C05474=1017.752,-121.815,388.715,-23.943,21.711,-44.591
C05475=1017.748,-122.143,388.737,-23.942,21.712,-44.597
C05476=1017.744,-122.471,388.759,-23.942,21.713,-44.601
C05477=1017.741,-122.799,388.781,-23.941,21.713,-44.606
C05478=1017.737,-123.128,388.803,-23.940,21.714,-44.610
C05479=1017.733,-123.456,388.826,-23.940,21.714,-44.615
C05480=1017.729,-123.785,388.848,-23.939,21.715,-44.620
C05481=1017.725,-124.112,388.871,-23.939,21.715,-44.625
C05482=1017.721,-124.441,388.893,-23.938,21.716,-44.628
C05483=1017.717,-124.769,388.915,-23.937,21.717,-44.634
C05484=1017.713,-125.097,388.937,-23.937,21.717,-44.638
C05485=1017.709,-125.425,388.959,-23.936,21.717,-44.643
C05486=1017.706,-125.754,388.981,-23.936,21.719,-44.647
C05487=1017.702,-126.082,389.003,-23.935,21.719,-44.652
C05488=1017.697,-126.409,389.026,-23.935,21.720,-44.657
C05489=1017.693,-126.737,389.048,-23.934,21.720,-44.662
C05490=1017.689,-127.066,389.070,-23.933,21.720,-44.667
C05491=1017.686,-127.394,389.092,-23.933,21.721,-44.671
C05492=1017.682,-127.722,389.114,-23.932,21.721,-44.676
C05493=1017.677,-128.050,389.136,-23.931,21.722,-44.680
C05494=1017.674,-128.378,389.158,-23.931,21.723,-44.686
C05495=1017.670,-128.706,389.180,-23.930,21.723,-44.689
C05496=1017.665,-129.034,389.202,-23.929,21.723,-44.695
C05497=1017.661,-129.362,389.224,-23.929,21.725,-44.699
C05498=1017.657,-129.690,389.246,-23.928,21.724,-44.704
C05499=1017.653,-130.018,389.268,-23.928,21.726,-44.708
C05500=1017.649,-130.346,389.290,-23.927,21.726,-44.713
C05501=1017.644,-130.674,389.312,-23.927,21.726,-44.717
C05502=1017.641,-131.002,389.334,-23.926,21.727,-44.723
C05503=1017.636,-131.331,389.356,-23.926,21.728,-44.726
C05504=1017.632,-131.659,389.378,-23.925,21.728,-44.732
C05505=1017.627,-131.986,389.400,-23.924,21.729,-44.736
C05506=1017.622,-132.314,389.422,-23.924,21.729,-44.741
C05507=1017.619,-132.643,389.444,-23.923,21.730,-44.745
C05508=1017.614,-132.971,389.465,-23.922,21.731,-44.750
C05509=1017.610,-133.299,389.488,-23.922,21.731,-44.754
C05510=1017.606,-133.626,389.510,-23.921,21.731,-44.759
C05511=1017.601,-133.954,389.531,-23.921,21.732,-44.763
C05512=1017.986,-133.926,389.292,-23.921,21.732,-44.763
C05513=1017.990,-133.599,389.270,-23.921,21.731,-44.759
C05514=1017.994,-133.271,389.248,-23.922,21.731,-44.754
C05515=1017.999,-132.943,389.226,-23.922,21.731,-44.750
C05516=1018.002,-132.614,389.204,-23.923,21.730,-44.745
C05517=1018.007,-132.287,389.182,-23.924,21.729,-44.741
C05518=1018.011,-131.959,389.161,-23.924,21.729,-44.736
C05519=1018.015,-131.630,389.139,-23.925,21.728,-44.732
C05520=1018.020,-131.303,389.117,-23.926,21.728,-44.726
C05521=1018.024,-130.975,389.094,-23.926,21.727,-44.723
C05522=1018.028,-130.647,389.073,-23.927,21.726,-44.717
C05523=1018.032,-130.319,389.051,-23.927,21.726,-44.713
C05524=1018.036,-129.990,389.029,-23.928,21.726,-44.708
C05525=1018.040,-129.662,389.007,-23.928,21.724,-44.704
C05526=1018.044,-129.334,388.985,-23.929,21.725,-44.699
C05527=1018.049,-129.006,388.964,-23.929,21.723,-44.695
C05528=1018.053,-128.679,388.941,-23.930,21.723,-44.689
C05529=1018.057,-128.350,388.919,-23.931,21.723,-44.686
C05530=1018.060,-128.022,388.897,-23.931,21.722,-44.680
C05531=1018.065,-127.694,388.875,-23.932,21.721,-44.676
C05532=1018.068,-127.367,388.853,-23.933,21.721,-44.671
C05533=1018.072,-127.038,388.831,-23.933,21.720,-44.667
C05534=1018.076,-126.710,388.809,-23.934,21.720,-44.662
C05535=1018.080,-126.382,388.788,-23.935,21.720,-44.657
C05536=1018.084,-126.054,388.766,-23.935,21.719,-44.652
C05537=1018.088,-125.726,388.743,-23.936,21.719,-44.647
C05538=1018.092,-125.398,388.721,-23.936,21.717,-44.643
C05539=1018.095,-125.070,388.699,-23.937,21.717,-44.638
C05540=1018.099,-124.741,388.676,-23.937,21.717,-44.634
C05541=1018.103,-124.413,388.654,-23.938,21.716,-44.628
C05542=1018.107,-124.085,388.632,-23.939,21.715,-44.625
C05543=1018.111,-123.757,388.610,-23.939,21.715,-44.620
C05544=1018.114,-123.428,388.588,-23.940,21.714,-44.615
C05545=1018.118,-123.100,388.566,-23.940,21.714,-44.610
C05546=1018.122,-122.772,388.544,-23.941,21.713,-44.606
C05547=1018.126,-122.444,388.522,-23.942,21.713,-44.601
C05548=1018.129,-122.115,388.500,-23.942,21.712,-44.597
C05549=1018.132,-121.787,388.477,-23.943,21.711,-44.591
C05550=1018.136,-121.459,388.455,-23.944,21.711,-44.586
C05551=1018.140,-121.130,388.433,-23.944,21.710,-44.582
C05552=1018.144,-120.802,388.411,-23.945,21.710,-44.577
C05553=1018.148,-120.474,388.389,-23.945,21.709,-44.573
C05554=1018.151,-120.145,388.366,-23.946,21.709,-44.568
C05555=1018.154,-119.817,388.344,-23.946,21.708,-44.564
C05556=1018.158,-119.489,388.322,-23.947,21.707,-44.558
C05557=1018.161,-119.160,388.299,-23.948,21.707,-44.554
C05558=1018.165,-118.832,388.277,-23.948,21.707,-44.549
C05559=1018.169,-118.504,388.255,-23.949,21.705,-44.545
C05560=1018.172,-118.175,388.232,-23.949,21.705,-44.540
C05561=1018.175,-117.847,388.210,-23.950,21.705,-44.535
C05562=1018.179,-117.518,388.187,-23.951,21.704,-44.531
C05563=1018.182,-117.190,388.165,-23.951,21.704,-44.525
C05564=1018.185,-116.862,388.142,-23.952,21.703,-44.521
C05565=1018.189,-116.533,388.120,-23.953,21.703,-44.516
C05566=1018.192,-116.205,388.098,-23.953,21.701,-44.512
C05567=1018.196,-115.876,388.076,-23.954,21.701,-44.507
C05568=1018.199,-115.548,388.053,-23.954,21.701,-44.503
C05569=1018.202,-115.219,388.030,-23.955,21.700,-44.497
C05570=1018.206,-114.891,388.008,-23.956,21.700,-44.492
C05571=1018.209,-114.562,387.985,-23.956,21.699,-44.488
C05572=1018.212,-114.234,387.963,-23.957,21.699,-44.483
C05573=1018.215,-113.905,387.940,-23.957,21.698,-44.479
C05574=1018.218,-113.576,387.919,-23.958,21.697,-44.473
C05575=1018.221,-113.248,387.896,-23.958,21.697,-44.470
C05576=1018.224,-112.919,387.873,-23.959,21.696,-44.464
C05577=1018.228,-112.590,387.850,-23.960,21.696,-44.459
C05578=1018.231,-112.261,387.827,-23.960,21.695,-44.455
C05579=1018.234,-111.933,387.805,-23.961,21.695,-44.449
C05580=1018.237,-111.604,387.782,-23.962,21.694,-44.446
C05581=1018.241,-111.276,387.760,-23.962,21.693,-44.440
C05582=1018.244,-110.947,387.738,-23.963,21.693,-44.436
C05583=1018.247,-110.618,387.715,-23.963,21.692,-44.431
C05584=1018.250,-110.289,387.692,-23.964,21.692,-44.426
C05585=1018.253,-109.960,387.669,-23.965,21.691,-44.422
C05586=1018.256,-109.632,387.646,-23.965,21.691,-44.416
C05587=1018.258,-109.302,387.624,-23.966,21.690,-44.412
C05588=1018.261,-108.974,387.602,-23.967,21.689,-44.407
C05589=1018.265,-108.645,387.578,-23.967,21.689,-44.402
C05590=1018.268,-108.316,387.556,-23.968,21.689,-44.398
C05591=1018.270,-107.987,387.532,-23.969,21.688,-44.392
C05592=1018.273,-107.658,387.511,-23.969,21.687,-44.388
C05593=1018.276,-107.329,387.488,-23.970,21.687,-44.383
C05594=1018.280,-107.000,387.465,-23.971,21.687,-44.378
C05595=1018.282,-106.671,387.441,-23.971,21.685,-44.374
C05596=1018.285,-106.342,387.419,-23.972,21.685,-44.368
C05597=1018.288,-106.013,387.397,-23.972,21.685,-44.365
C05598=1018.291,-105.684,387.373,-23.973,21.684,-44.359
C05599=1018.294,-105.355,387.350,-23.974,21.684,-44.354
C05600=1018.296,-105.027,387.328,-23.974,21.683,-44.350
C05601=1018.299,-104.699,387.305,-23.975,21.683,-44.344
C05602=1018.302,-104.370,387.282,-23.975,21.681,-44.340
C05603=1018.304,-104.043,387.259,-23.976,21.681,-44.335
C05604=1018.308,-103.716,387.237,-23.976,21.681,-44.331
C05605=1018.310,-103.389,387.214,-23.977,21.680,-44.326
C05606=1018.313,-103.062,387.191,-23.978,21.680,-44.320
C05607=1018.316,-102.736,387.169,-23.978,21.679,-44.316
C05608=1018.317,-102.411,387.146,-23.979,21.679,-44.311
C05609=1018.321,-102.085,387.123,-23.980,21.678,-44.307
C05610=1018.323,-101.762,387.100,-23.980,21.677,-44.302
C05611=1018.325,-101.437,387.078,-23.981,21.677,-44.298
C05612=1018.328,-101.113,387.055,-23.981,21.676,-44.292
C05613=1018.331,-100.790,387.033,-23.982,21.676,-44.287
C05614=1018.333,-100.468,387.010,-23.983,21.675,-44.283
C05615=1018.336,-100.146,386.987,-23.983,21.675,-44.278
C05616=1018.338,-99.824,386.965,-23.984,21.674,-44.274
C05617=1018.341,-99.502,386.942,-23.985,21.673,-44.268
C05618=1018.343,-99.181,386.920,-23.985,21.673,-44.265
C05619=1018.345,-98.860,386.898,-23.986,21.673,-44.260
C05620=1018.348,-98.539,386.874,-23.986,21.671,-44.255
C05621=1018.351,-98.217,386.852,-23.987,21.672,-44.250
C05622=1018.353,-97.897,386.829,-23.987,21.670,-44.246
C05623=1018.355,-97.576,386.807,-23.988,21.670,-44.241
C05624=1018.358,-97.255,386.784,-23.989,21.670,-44.236
C05625=1018.360,-96.934,386.762,-23.989,21.669,-44.231
C05626=1018.361,-96.613,386.739,-23.990,21.669,-44.226
C05627=1018.364,-96.291,386.716,-23.991,21.668,-44.222
C05628=1018.366,-95.970,386.694,-23.991,21.668,-44.217
C05629=1018.368,-95.648,386.671,-23.992,21.667,-44.213
C05630=1018.371,-95.326,386.648,-23.993,21.666,-44.207
C05631=1018.373,-95.003,386.626,-23.993,21.666,-44.204
C05632=1018.375,-94.680,386.603,-23.994,21.666,-44.199
C05633=1018.378,-94.357,386.580,-23.994,21.665,-44.193
C05634=1018.380,-94.032,386.557,-23.995,21.664,-44.189
C05635=1018.382,-93.708,386.534,-23.996,21.664,-44.184
C05636=1018.384,-93.382,386.510,-23.996,21.663,-44.180
C05637=1018.386,-93.057,386.487,-23.997,21.663,-44.175
C05638=1018.388,-92.731,386.465,-23.998,21.662,-44.169
C05639=1018.391,-92.405,386.441,-23.998,21.662,-44.165
C05640=1018.392,-92.077,386.418,-23.999,21.661,-44.160
C05641=1018.395,-91.749,386.395,-23.999,21.660,-44.156
C05642=1018.398,-91.420,386.372,-24.000,21.660,-44.150
C05643=1018.398,-91.092,386.349,-24.001,21.660,-44.145
C05644=1018.401,-90.762,386.325,-24.001,21.659,-44.141
C05645=1018.404,-90.433,386.302,-24.002,21.658,-44.136
C05646=1018.406,-90.095,386.277,-24.003,21.658,-44.130
C05647=1018.408,-89.689,386.249,-24.004,21.657,-44.123
C05648=1018.410,-89.459,386.232,-24.004,21.656,-44.121
C05649=1018.411,-89.220,386.215,-24.004,21.656,-44.119
C05650=1018.412,-88.986,386.199,-24.004,21.656,-44.117
C05651=1018.414,-88.768,386.183,-24.005,21.656,-44.114
C05652=1018.416,-88.396,386.156,-24.006,21.655,-44.106
C05653=1018.418,-88.077,386.134,-24.006,21.654,-44.102
C05654=1018.420,-87.765,386.111,-24.007,21.654,-44.097
C05655=1018.421,-87.454,386.089,-24.007,21.653,-44.093
C05656=1018.423,-87.142,386.066,-24.008,21.653,-44.088
C05657=1018.425,-86.826,386.044,-24.009,21.652,-44.082
C05658=1018.427,-86.503,386.021,-24.009,21.652,-44.078
C05659=1018.430,-86.174,385.997,-24.010,21.651,-44.073
C05660=1018.431,-85.814,385.971,-24.011,21.650,-44.067
C05661=1018.433,-85.405,385.942,-24.012,21.649,-44.062
C05662=1018.434,-85.193,385.927,-24.012,21.649,-44.060
C05663=1018.436,-84.980,385.912,-24.012,21.650,-44.056
C05664=1018.438,-84.583,385.883,-24.013,21.649,-44.051
C05665=1018.439,-84.233,385.858,-24.014,21.648,-44.045
C05666=1018.441,-83.899,385.834,-24.015,21.648,-44.040
C05667=1018.443,-83.564,385.809,-24.015,21.647,-44.036
C05668=1018.445,-83.229,385.786,-24.016,21.647,-44.031
C05669=1018.447,-82.893,385.762,-24.016,21.646,-44.025
C05670=1018.448,-82.557,385.737,-24.017,21.645,-44.021
C05671=1018.450,-82.221,385.713,-24.018,21.645,-44.016
C05672=1018.451,-81.883,385.689,-24.018,21.645,-44.010
C05673=1018.453,-81.546,385.664,-24.019,21.644,-44.005
C05674=1018.456,-81.208,385.640,-24.020,21.643,-44.001
C05675=1018.456,-80.870,385.616,-24.020,21.643,-43.995
C05676=1018.458,-80.532,385.591,-24.021,21.643,-43.990
C05677=1018.460,-80.192,385.567,-24.021,21.641,-43.986
C05678=1018.462,-79.853,385.541,-24.022,21.641,-43.981
C05679=1018.463,-79.513,385.517,-24.023,21.641,-43.975
C05680=1018.464,-79.173,385.492,-24.023,21.639,-43.971
C05681=1018.466,-78.833,385.467,-24.024,21.639,-43.966
C05682=1018.468,-78.492,385.443,-24.025,21.638,-43.960
C05683=1018.470,-78.150,385.418,-24.026,21.639,-43.955
C05684=1018.472,-77.809,385.394,-24.026,21.637,-43.951
C05685=1018.473,-77.468,385.368,-24.027,21.637,-43.946
C05686=1018.474,-77.125,385.343,-24.028,21.636,-43.940
C05687=1018.476,-76.783,385.319,-24.028,21.636,-43.936
C05688=1018.478,-76.441,385.294,-24.029,21.635,-43.931
C05689=1018.479,-76.098,385.269,-24.030,21.635,-43.926
C05690=1018.480,-75.755,385.244,-24.030,21.634,-43.920
C05691=1018.482,-75.412,385.219,-24.031,21.634,-43.916
C05692=1018.482,-75.069,385.194,-24.031,21.633,-43.911
C05693=1018.484,-74.725,385.169,-24.032,21.633,-43.905
C05694=1018.486,-74.383,385.144,-24.033,21.632,-43.901
C05695=1018.487,-74.039,385.118,-24.033,21.632,-43.896
C05696=1018.489,-73.695,385.093,-24.034,21.631,-43.890
C05697=1018.489,-73.351,385.068,-24.035,21.630,-43.885
C05698=1018.491,-73.008,385.043,-24.035,21.630,-43.881
C05699=1018.493,-72.664,385.017,-24.036,21.629,-43.875
C05700=1018.494,-72.319,384.992,-24.037,21.629,-43.870
C05701=1018.496,-71.975,384.967,-24.038,21.628,-43.865
C05702=1018.496,-71.632,384.942,-24.038,21.628,-43.861
C05703=1018.497,-71.288,384.917,-24.039,21.627,-43.855
C05704=1018.498,-70.944,384.891,-24.040,21.627,-43.850
C05705=1018.500,-70.599,384.866,-24.040,21.626,-43.844
C05706=1018.501,-70.250,384.840,-24.041,21.625,-43.840
C05707=1018.502,-69.911,384.815,-24.041,21.625,-43.835
C05708=1018.503,-69.567,384.790,-24.042,21.624,-43.829
C05709=1018.505,-69.223,384.764,-24.043,21.624,-43.824
C05710=1018.505,-68.879,384.739,-24.043,21.623,-43.820
C05711=1018.507,-68.535,384.714,-24.044,21.623,-43.815
C05712=1018.508,-68.192,384.688,-24.045,21.622,-43.809
C05713=1018.509,-67.848,384.663,-24.045,21.622,-43.805
C05714=1018.510,-67.504,384.637,-24.046,21.621,-43.800
C05715=1018.511,-67.161,384.612,-24.047,21.621,-43.795
C05716=1018.512,-66.818,384.587,-24.048,21.620,-43.789
C05717=1018.513,-66.475,384.562,-24.048,21.620,-43.785
C05718=1018.514,-66.132,384.535,-24.049,21.619,-43.780
C05719=1018.515,-65.789,384.511,-24.050,21.619,-43.774
C05720=1018.516,-65.448,384.485,-24.050,21.617,-43.770
C05721=1018.517,-65.105,384.459,-24.051,21.618,-43.765
C05722=1018.518,-64.764,384.434,-24.051,21.617,-43.759
C05723=1018.519,-64.422,384.408,-24.052,21.617,-43.754
C05724=1018.520,-64.080,384.383,-24.053,21.615,-43.750
C05725=1018.521,-63.740,384.358,-24.053,21.616,-43.745
C05726=1018.521,-63.399,384.333,-24.054,21.615,-43.739
C05727=1018.522,-63.059,384.308,-24.055,21.614,-43.735
C05728=1018.523,-62.719,384.282,-24.055,21.613,-43.730
C05729=1018.525,-62.379,384.256,-24.056,21.614,-43.725
C05730=1018.525,-62.040,384.231,-24.057,21.612,-43.720
C05731=1018.526,-61.701,384.206,-24.057,21.612,-43.715
C05732=1018.526,-61.363,384.181,-24.058,21.611,-43.710
C05733=1018.527,-61.024,384.155,-24.059,21.611,-43.706
C05734=1018.528,-60.687,384.130,-24.059,21.610,-43.700
C05735=1018.528,-60.350,384.105,-24.060,21.610,-43.695
C05736=1018.529,-60.013,384.080,-24.060,21.609,-43.691
C05737=1018.530,-59.677,384.055,-24.061,21.609,-43.686
C05738=1018.531,-59.341,384.029,-24.062,21.608,-43.680
C05739=1018.531,-59.005,384.004,-24.062,21.608,-43.676
C05740=1018.532,-58.670,383.979,-24.063,21.607,-43.671
C05741=1018.532,-58.335,383.954,-24.064,21.607,-43.666
C05742=1018.533,-58.000,383.929,-24.064,21.606,-43.662
C05743=1018.534,-57.666,383.903,-24.065,21.606,-43.656
C05744=1018.535,-57.332,383.879,-24.066,21.605,-43.652
C05745=1018.535,-56.998,383.853,-24.066,21.604,-43.647
C05746=1018.536,-56.665,383.828,-24.067,21.605,-43.642
C05747=1018.536,-56.332,383.803,-24.068,21.603,-43.637
C05748=1018.537,-55.999,383.778,-24.068,21.603,-43.632
C05749=1018.537,-55.667,383.753,-24.069,21.603,-43.627
C05750=1018.537,-55.334,383.728,-24.070,21.602,-43.623
C05751=1018.539,-55.001,383.702,-24.070,21.602,-43.618
C05752=1018.538,-54.668,383.677,-24.071,21.601,-43.613
C05753=1018.539,-54.336,383.652,-24.072,21.601,-43.608
C05754=1018.539,-54.004,383.627,-24.072,21.600,-43.603
C05755=1018.540,-53.672,383.602,-24.073,21.599,-43.599
C05756=1018.541,-53.339,383.576,-24.074,21.600,-43.594
C05757=1018.540,-53.007,383.551,-24.074,21.598,-43.589
C05758=1018.541,-52.675,383.526,-24.075,21.598,-43.584
C05759=1018.541,-52.342,383.501,-24.075,21.597,-43.579
C05760=1018.542,-52.010,383.476,-24.076,21.597,-43.575
C05761=1018.543,-51.678,383.451,-24.077,21.597,-43.570
C05762=1018.542,-51.345,383.426,-24.077,21.596,-43.566
C05763=1018.543,-51.013,383.400,-24.078,21.596,-43.560
C05764=1018.544,-50.681,383.375,-24.079,21.595,-43.555
C05765=1018.544,-50.348,383.350,-24.079,21.594,-43.551
C05766=1018.544,-50.016,383.324,-24.080,21.595,-43.546
C05767=1018.544,-49.684,383.298,-24.080,21.593,-43.542
C05768=1018.544,-49.351,383.273,-24.081,21.593,-43.536
C05769=1018.545,-49.019,383.248,-24.081,21.592,-43.532
C05770=1018.545,-48.686,383.223,-24.082,21.592,-43.527
C05771=1018.545,-48.354,383.198,-24.083,21.592,-43.522
C05772=1018.545,-48.022,383.172,-24.083,21.591,-43.518
C05773=1018.545,-47.689,383.147,-24.084,21.591,-43.512
C05774=1018.545,-47.357,383.121,-24.085,21.589,-43.508
C05775=1018.545,-47.024,383.096,-24.086,21.589,-43.503
C05776=1018.546,-46.692,383.071,-24.086,21.590,-43.498
C05777=1018.546,-46.360,383.045,-24.087,21.588,-43.494
C05778=1018.546,-46.027,383.020,-24.088,21.588,-43.488
C05779=1018.546,-45.695,382.994,-24.088,21.588,-43.485
C05780=1018.545,-45.361,382.969,-24.089,21.587,-43.479
C05781=1018.546,-45.028,382.943,-24.089,21.586,-43.475
C05782=1018.546,-44.696,382.917,-24.090,21.586,-43.470
C05783=1018.546,-44.363,382.892,-24.091,21.586,-43.465
C05784=1018.546,-44.031,382.866,-24.091,21.585,-43.461
C05785=1018.546,-43.699,382.840,-24.092,21.585,-43.455
C05786=1018.546,-43.366,382.815,-24.092,21.584,-43.451
C05787=1018.546,-43.034,382.789,-24.093,21.583,-43.446
C05788=1018.546,-42.701,382.764,-24.094,21.583,-43.442
C05789=1018.545,-42.368,382.738,-24.094,21.583,-43.437
C05790=1018.546,-42.036,382.713,-24.095,21.582,-43.431
C05791=1018.546,-41.703,382.688,-24.096,21.582,-43.427
C05792=1018.545,-41.371,382.661,-24.096,21.582,-43.422
C05793=1018.545,-41.039,382.636,-24.097,21.580,-43.418
C05794=1018.546,-40.705,382.610,-24.098,21.580,-43.413
C05795=1018.545,-40.373,382.584,-24.098,21.580,-43.409
C05796=1018.546,-40.040,382.558,-24.099,21.579,-43.404
C05797=1018.545,-39.707,382.533,-24.100,21.579,-43.398
C05798=1018.545,-39.375,382.507,-24.100,21.578,-43.394
C05799=1018.544,-39.043,382.481,-24.101,21.578,-43.389
C05800=1018.544,-38.710,382.456,-24.101,21.577,-43.385
C05801=1018.544,-38.377,382.429,-24.102,21.577,-43.380
C05802=1018.544,-38.045,382.404,-24.102,21.576,-43.376
C05803=1018.543,-37.712,382.378,-24.103,21.576,-43.371
C05804=1018.543,-37.379,382.352,-24.104,21.575,-43.366
C05805=1018.544,-37.046,382.326,-24.105,21.575,-43.361
C05806=1018.543,-36.713,382.300,-24.105,21.574,-43.357
C05807=1018.542,-36.381,382.274,-24.106,21.574,-43.352
C05808=1018.542,-36.049,382.248,-24.107,21.574,-43.347
C05809=1018.542,-35.715,382.223,-24.107,21.573,-43.343
C05810=1018.541,-35.383,382.196,-24.108,21.573,-43.337
C05811=1018.541,-35.051,382.171,-24.108,21.572,-43.334
C05812=1018.541,-34.718,382.145,-24.109,21.572,-43.328
C05813=1018.540,-34.385,382.119,-24.109,21.571,-43.324
C05814=1018.540,-34.053,382.093,-24.110,21.571,-43.319
C05815=1018.539,-33.720,382.066,-24.111,21.570,-43.315
C05816=1018.539,-33.387,382.041,-24.111,21.570,-43.310
C05817=1018.539,-33.054,382.015,-24.112,21.569,-43.306
C05818=1018.539,-32.721,381.988,-24.113,21.569,-43.301
C05819=1018.538,-32.388,381.963,-24.113,21.568,-43.296
C05820=1018.537,-32.056,381.937,-24.114,21.568,-43.291
C05821=1018.537,-31.723,381.910,-24.114,21.567,-43.287
C05822=1018.536,-31.391,381.884,-24.115,21.567,-43.282
C05823=1018.535,-31.058,381.858,-24.116,21.566,-43.278
C05824=1018.535,-30.725,381.832,-24.116,21.566,-43.273
C05825=1018.534,-30.393,381.806,-24.117,21.565,-43.269
C05826=1018.534,-30.060,381.780,-24.118,21.565,-43.264
C05827=1018.533,-29.727,381.754,-24.118,21.565,-43.260
C05828=1018.533,-29.394,381.728,-24.119,21.564,-43.254
C05829=1018.533,-29.061,381.701,-24.119,21.563,-43.250
C05830=1018.532,-28.729,381.675,-24.120,21.563,-43.245
C05831=1018.531,-28.396,381.649,-24.120,21.562,-43.241
C05832=1018.530,-28.063,381.622,-24.121,21.562,-43.236
C05833=1018.530,-27.730,381.596,-24.122,21.562,-43.232
C05834=1018.529,-27.398,381.570,-24.123,21.562,-43.227
C05835=1018.528,-27.065,381.544,-24.123,21.560,-43.223
C05836=1018.528,-26.732,381.518,-24.124,21.560,-43.217
C05837=1018.526,-26.399,381.491,-24.124,21.560,-43.214
C05838=1018.526,-26.067,381.465,-24.125,21.559,-43.208
C05839=1018.525,-25.734,381.438,-24.126,21.559,-43.204
C05840=1018.525,-25.401,381.413,-24.126,21.559,-43.199
C05841=1018.523,-25.068,381.386,-24.127,21.558,-43.195
C05842=1018.523,-24.736,381.360,-24.128,21.558,-43.190
C05843=1018.522,-24.403,381.333,-24.128,21.557,-43.186
C05844=1018.521,-24.070,381.307,-24.129,21.557,-43.181
C05845=1018.520,-23.737,381.281,-24.129,21.556,-43.177
C05846=1018.520,-23.404,381.254,-24.130,21.556,-43.171
C05847=1018.519,-23.071,381.228,-24.131,21.555,-43.168
C05848=1018.518,-22.738,381.201,-24.131,21.556,-43.162
C05849=1018.517,-22.406,381.174,-24.132,21.554,-43.158
C05850=1018.516,-22.072,381.148,-24.133,21.554,-43.153
C05851=1018.515,-21.740,381.122,-24.133,21.554,-43.149
C05852=1018.514,-21.407,381.095,-24.134,21.553,-43.144
C05853=1018.514,-21.074,381.069,-24.134,21.552,-43.140
C05854=1018.512,-20.742,381.042,-24.135,21.553,-43.135
C05855=1018.512,-20.409,381.016,-24.136,21.552,-43.131
C05856=1018.511,-20.076,380.989,-24.136,21.551,-43.127
C05857=1018.510,-19.743,380.963,-24.137,21.551,-43.122
C05858=1018.509,-19.571,380.949,-24.137,21.550,-43.118
C05859=1018.507,-19.155,380.915,-24.138,21.550,-43.112
C05860=1018.507,-18.907,380.896,-24.139,21.550,-43.109
C05861=1018.506,-18.645,380.875,-24.139,21.550,-43.107
C05862=1018.505,-18.383,380.854,-24.139,21.549,-43.105
C05863=1018.504,-18.136,380.834,-24.139,21.548,-43.103
C05864=1018.504,-17.914,380.817,-24.140,21.549,-43.100
C05865=1018.502,-17.549,380.787,-24.141,21.548,-43.092
C05866=1018.502,-17.216,380.761,-24.141,21.547,-43.088
C05867=1018.501,-16.884,380.734,-24.142,21.547,-43.083
C05868=1018.499,-16.550,380.708,-24.142,21.547,-43.079
C05869=1018.498,-16.217,380.680,-24.143,21.546,-43.074
C05870=1018.497,-15.882,380.653,-24.144,21.546,-43.070
C05871=1018.495,-15.546,380.626,-24.145,21.546,-43.065
C05872=1018.495,-15.210,380.599,-24.145,21.545,-43.061
C05873=1018.493,-14.873,380.573,-24.146,21.544,-43.055
C05874=1018.492,-14.532,380.545,-24.146,21.544,-43.052
C05875=1018.491,-14.191,380.518,-24.147,21.544,-43.046
C05876=1018.490,-13.846,380.490,-24.147,21.543,-43.042
C05877=1018.489,-13.499,380.462,-24.148,21.543,-43.037
C05878=1018.487,-13.151,380.434,-24.149,21.542,-43.033
C05879=1018.486,-12.801,380.406,-24.149,21.542,-43.028
C05880=1018.484,-12.449,380.378,-24.150,21.541,-43.024
C05881=1018.483,-12.096,380.349,-24.151,21.541,-43.019
C05882=1018.482,-11.740,380.320,-24.151,21.540,-43.014
C05883=1018.480,-11.384,380.292,-24.152,21.540,-43.009
C05884=1018.479,-11.026,380.262,-24.152,21.539,-43.006
C05885=1018.477,-10.667,380.233,-24.153,21.539,-43.000
C05886=1018.476,-10.307,380.204,-24.154,21.539,-42.995
C05887=1018.474,-9.947,380.175,-24.154,21.538,-42.991
C05888=1018.473,-9.584,380.146,-24.155,21.538,-42.985
C05889=1018.471,-9.223,380.116,-24.156,21.537,-42.982
C05890=1018.470,-8.861,380.087,-24.156,21.536,-42.976
C05891=1018.468,-8.498,380.057,-24.157,21.536,-42.971
C05892=1018.466,-8.135,380.029,-24.158,21.536,-42.967
C05893=1018.464,-7.761,379.998,-24.158,21.535,-42.961
C05894=1018.463,-7.405,379.969,-24.159,21.535,-42.956
C05895=1018.462,-7.036,379.939,-24.160,21.534,-42.952
C05896=1018.460,-6.664,379.909,-24.160,21.534,-42.947
C05897=1018.458,-6.290,379.879,-24.161,21.533,-42.941
C05898=1018.457,-5.914,379.848,-24.162,21.533,-42.937
C05899=1018.455,-5.539,379.817,-24.163,21.533,-42.932
C05900=1018.453,-5.165,379.786,-24.163,21.532,-42.928
C05901=1018.450,-4.795,379.757,-24.164,21.532,-42.923
C05902=1018.449,-4.428,379.727,-24.164,21.531,-42.919
C05903=1018.447,-4.067,379.697,-24.165,21.530,-42.913
C05904=1018.446,-3.710,379.668,-24.166,21.531,-42.908
C05905=1018.444,-3.355,379.639,-24.166,21.529,-42.904
C05906=1018.442,-3.003,379.610,-24.167,21.529,-42.899
C05907=1018.440,-2.651,379.582,-24.167,21.529,-42.895
C05908=1018.439,-2.302,379.553,-24.168,21.529,-42.890
C05909=1018.437,-1.953,379.524,-24.169,21.528,-42.886
C05910=1018.435,-1.607,379.496,-24.169,21.528,-42.880
C05911=1018.433,-1.262,379.469,-24.170,21.527,-42.877
C05912=1018.431,-0.919,379.439,-24.170,21.527,-42.873
C05913=1018.429,-0.577,379.412,-24.171,21.526,-42.867
C05914=1018.428,-0.237,379.384,-24.172,21.526,-42.864
C05915=1018.426,0.102,379.356,-24.172,21.526,-42.858
C05916=1018.424,0.439,379.328,-24.173,21.525,-42.855
C05917=1018.422,0.775,379.300,-24.173,21.525,-42.851
C05918=1018.421,1.109,379.273,-24.174,21.525,-42.846
C05919=1018.418,1.444,379.246,-24.175,21.524,-42.842
C05920=1018.416,1.777,379.218,-24.175,21.523,-42.838
C05921=1018.415,2.108,379.192,-24.176,21.523,-42.834
C05922=1018.413,2.420,379.165,-24.176,21.523,-42.831
C05923=1018.411,2.708,379.142,-24.177,21.522,-42.827
C05924=1018.410,2.977,379.120,-24.177,21.522,-42.823
C05925=1018.408,3.239,379.098,-24.178,21.522,-42.818
C05926=1018.407,3.509,379.076,-24.179,21.521,-42.814
C05927=1018.405,3.798,379.053,-24.179,21.521,-42.810
C05928=1018.403,4.111,379.026,-24.179,21.520,-42.807
C05929=1018.401,4.440,378.999,-24.180,21.521,-42.803
C05930=1018.399,4.772,378.971,-24.180,21.519,-42.799
C05931=1018.397,5.103,378.944,-24.181,21.519,-42.795
C05932=1018.395,5.434,378.918,-24.181,21.518,-42.792
C05933=1018.393,5.764,378.890,-24.182,21.519,-42.786
C05934=1018.391,6.094,378.862,-24.183,21.518,-42.783
C05935=1018.389,6.424,378.835,-24.183,21.518,-42.779
C05936=1018.387,6.753,378.809,-24.184,21.518,-42.774
C05937=1018.385,7.081,378.781,-24.185,21.517,-42.770
C05938=1018.383,7.409,378.754,-24.185,21.517,-42.766
C05939=1018.381,7.734,378.727,-24.186,21.516,-42.762
C05940=1018.378,8.057,378.700,-24.186,21.516,-42.759
C05941=1018.377,8.378,378.673,-24.186,21.515,-42.755
C05942=1018.375,8.696,378.647,-24.187,21.516,-42.750
C05943=1018.373,9.013,378.621,-24.188,21.515,-42.746
C05944=1018.370,9.328,378.595,-24.188,21.515,-42.742
C05945=1018.369,9.642,378.568,-24.189,21.514,-42.738
C05946=1018.366,9.958,378.542,-24.190,21.514,-42.733
C05947=1018.364,10.273,378.517,-24.190,21.514,-42.730
C05948=1018.362,10.590,378.489,-24.191,21.513,-42.726
C05949=1018.360,10.908,378.463,-24.191,21.513,-42.722
C05950=1018.358,11.229,378.437,-24.192,21.512,-42.718
C05951=1018.355,11.552,378.410,-24.192,21.512,-42.715
C05952=1018.354,11.875,378.383,-24.193,21.511,-42.711
C05953=1018.351,12.198,378.356,-24.193,21.511,-42.707
C05954=1018.349,12.522,378.329,-24.194,21.511,-42.702
C05955=1018.347,12.845,378.302,-24.194,21.510,-42.698
C05956=1018.344,13.169,378.275,-24.195,21.510,-42.694
C05957=1018.342,13.493,378.248,-24.195,21.509,-42.691
C05958=1018.340,13.817,378.221,-24.196,21.509,-42.687
C05959=1018.338,14.142,378.194,-24.197,21.509,-42.682
C05960=1018.335,14.466,378.167,-24.197,21.509,-42.678
C05961=1018.333,14.791,378.140,-24.198,21.508,-42.674
C05962=1018.330,15.117,378.113,-24.198,21.508,-42.670
C05963=1018.328,15.442,378.085,-24.199,21.507,-42.667
C05964=1018.326,15.769,378.057,-24.199,21.507,-42.663
C05965=1018.323,16.096,378.031,-24.200,21.507,-42.658
C05966=1018.321,16.423,378.003,-24.200,21.506,-42.654
C05967=1018.319,16.751,377.976,-24.201,21.506,-42.650
C05968=1018.316,17.081,377.948,-24.201,21.505,-42.646
C05969=1018.314,17.409,377.920,-24.202,21.505,-42.643
C05970=1018.311,17.739,377.893,-24.202,21.504,-42.639
C05971=1018.309,18.069,377.865,-24.203,21.504,-42.634
C05972=1018.306,18.400,377.838,-24.204,21.504,-42.630
C05973=1018.303,18.732,377.810,-24.204,21.503,-42.626
C05974=1018.301,19.063,377.782,-24.205,21.503,-42.622
C05975=1018.298,19.395,377.754,-24.205,21.502,-42.619
C05976=1018.296,19.743,377.725,-24.206,21.503,-42.613
C05977=1018.293,20.161,377.690,-24.207,21.502,-42.608
C05978=1018.290,20.397,377.670,-24.207,21.502,-42.604
C05979=1018.289,20.643,377.649,-24.207,21.502,-42.603
C05980=1018.286,20.892,377.628,-24.208,21.502,-42.601
C05981=1018.285,21.134,377.607,-24.208,21.502,-42.599
C05982=1018.283,21.361,377.589,-24.208,21.501,-42.597
C05983=1018.281,21.568,377.572,-24.209,21.501,-42.593
C05984=1018.279,21.925,377.541,-24.209,21.500,-42.588
C05985=1018.276,22.249,377.515,-24.210,21.501,-42.584
C05986=1018.273,22.543,377.489,-24.210,21.500,-42.582
C05987=1018.271,22.796,377.467,-24.210,21.499,-42.580
C05988=1018.268,23.206,377.434,-24.211,21.499,-42.573
C05989=1018.264,23.613,377.399,-24.212,21.498,-42.565
C05990=1018.263,23.865,377.378,-24.213,21.498,-42.562
C05991=1018.260,24.159,377.353,-24.213,21.498,-42.560
C05992=1018.257,24.486,377.325,-24.213,21.497,-42.558
C05993=1018.255,24.821,377.297,-24.214,21.497,-42.553
C05994=1018.252,25.154,377.269,-24.215,21.497,-42.549
C05995=1018.249,25.490,377.241,-24.215,21.496,-42.545
C05996=1018.247,25.824,377.212,-24.216,21.496,-42.541
C05997=1018.243,26.158,377.184,-24.216,21.495,-42.538
C05998=1018.241,26.492,377.156,-24.217,21.495,-42.534
C05999=1018.237,26.826,377.127,-24.217,21.494,-42.530
C06000=1018.234,27.161,377.099,-24.218,21.494,-42.525
C06001=1018.232,27.495,377.071,-24.219,21.495,-42.522
C06002=1018.228,27.830,377.043,-24.219,21.494,-42.518
C06003=1018.226,28.164,377.014,-24.220,21.494,-42.514
C06004=1018.223,28.499,376.986,-24.220,21.493,-42.510
C06005=1018.219,28.833,376.957,-24.221,21.493,-42.507
C06006=1018.217,29.168,376.929,-24.221,21.492,-42.503
C06007=1018.214,29.502,376.900,-24.222,21.493,-42.498
C06008=1018.210,29.837,376.872,-24.222,21.492,-42.494
C06009=1018.207,30.171,376.843,-24.223,21.492,-42.490
C06010=1018.205,30.506,376.816,-24.223,21.491,-42.486
C06011=1018.201,30.840,376.787,-24.224,21.491,-42.483
C06012=1018.199,31.174,376.758,-24.224,21.490,-42.479
C06013=1018.195,31.509,376.730,-24.225,21.490,-42.475
C06014=1018.192,31.844,376.702,-24.225,21.489,-42.471
C06015=1018.189,32.178,376.673,-24.226,21.489,-42.468
C06016=1018.186,32.513,376.645,-24.226,21.489,-42.464
C06017=1018.183,32.847,376.616,-24.227,21.489,-42.459
C06018=1018.180,33.182,376.588,-24.228,21.489,-42.455
C06019=1018.177,33.516,376.559,-24.228,21.488,-42.452
C06020=1018.174,33.851,376.531,-24.229,21.488,-42.448
C06021=1018.170,34.185,376.502,-24.229,21.487,-42.444
C06022=1018.167,34.520,376.474,-24.230,21.487,-42.440
C06023=1018.164,34.855,376.445,-24.230,21.486,-42.437
C06024=1018.160,35.189,376.417,-24.231,21.486,-42.433
C06025=1018.158,35.524,376.388,-24.231,21.485,-42.429
C06026=1018.154,35.859,376.359,-24.232,21.486,-42.426
C06027=1018.151,36.194,376.330,-24.232,21.485,-42.422
C06028=1018.147,36.528,376.302,-24.233,21.485,-42.418
C06029=1018.144,36.863,376.273,-24.234,21.485,-42.413
C06030=1018.141,37.198,376.244,-24.234,21.485,-42.409
C06031=1018.138,37.533,376.216,-24.235,21.484,-42.405
C06032=1018.134,37.867,376.187,-24.235,21.484,-42.402
C06033=1018.130,38.202,376.159,-24.236,21.483,-42.398
C06034=1018.128,38.536,376.130,-24.236,21.483,-42.395
C06035=1018.124,38.872,376.101,-24.237,21.483,-42.391
C06036=1018.120,39.206,376.073,-24.237,21.483,-42.387
C06037=1018.117,39.541,376.044,-24.238,21.482,-42.383
C06038=1018.114,39.876,376.015,-24.238,21.482,-42.380
C06039=1018.110,40.211,375.986,-24.239,21.481,-42.376
C06040=1018.106,40.545,375.958,-24.239,21.481,-42.372
C06041=1018.103,40.880,375.929,-24.240,21.481,-42.369
C06042=1018.100,41.215,375.900,-24.240,21.481,-42.365
C06043=1018.096,41.550,375.872,-24.241,21.480,-42.361
C06044=1018.092,41.884,375.842,-24.241,21.480,-42.357
C06045=1018.089,42.219,375.814,-24.242,21.479,-42.354
C06046=1018.085,42.555,375.785,-24.242,21.479,-42.350
C06047=1018.082,42.889,375.756,-24.243,21.479,-42.347
C06048=1018.078,43.225,375.727,-24.243,21.479,-42.343
C06049=1018.075,43.558,375.698,-24.244,21.478,-42.339
C06050=1018.071,43.894,375.670,-24.244,21.478,-42.335
C06051=1018.068,44.229,375.641,-24.245,21.477,-42.332
C06052=1018.064,44.564,375.612,-24.245,21.477,-42.328
C06053=1018.060,44.899,375.583,-24.246,21.477,-42.325
C06054=1018.057,45.234,375.555,-24.246,21.477,-42.321
C06055=1018.053,45.568,375.525,-24.247,21.476,-42.317
C06056=1018.050,45.904,375.497,-24.247,21.476,-42.313
C06057=1018.046,46.238,375.468,-24.248,21.475,-42.309
C06058=1018.042,46.573,375.439,-24.248,21.475,-42.306
C06059=1018.038,46.909,375.410,-24.249,21.475,-42.302
C06060=1018.035,47.243,375.381,-24.249,21.475,-42.299
C06061=1018.030,47.578,375.352,-24.250,21.474,-42.295
C06062=1018.026,47.913,375.323,-24.250,21.474,-42.291
C06063=1018.023,48.248,375.294,-24.251,21.473,-42.287
C06064=1018.020,48.583,375.265,-24.251,21.473,-42.284
C06065=1018.015,48.918,375.237,-24.252,21.473,-42.280
C06066=1018.011,49.253,375.207,-24.252,21.473,-42.277
C06067=1018.008,49.588,375.178,-24.253,21.472,-42.273
C06068=1018.004,49.923,375.149,-24.253,21.472,-42.269
C06069=1017.999,50.258,375.120,-24.254,21.472,-42.266
C06070=1017.996,50.593,375.091,-24.254,21.471,-42.262
C06071=1017.993,50.928,375.062,-24.255,21.471,-42.258
C06072=1017.988,51.262,375.034,-24.255,21.471,-42.254
C06073=1017.984,51.598,375.005,-24.256,21.471,-42.251
C06074=1017.981,51.932,374.975,-24.256,21.470,-42.247
C06075=1017.977,52.268,374.946,-24.257,21.470,-42.244
C06076=1017.972,52.603,374.918,-24.257,21.470,-42.240
C06077=1017.969,52.937,374.888,-24.258,21.469,-42.238
C06078=1017.965,53.273,374.859,-24.258,21.469,-42.234
C06079=1017.960,53.608,374.830,-24.259,21.468,-42.230
C06080=1017.957,53.942,374.801,-24.259,21.468,-42.227
C06081=1017.952,54.278,374.771,-24.260,21.468,-42.223
C06082=1017.948,54.612,374.742,-24.260,21.468,-42.220
C06083=1017.944,54.948,374.713,-24.261,21.467,-42.216
C06084=1017.940,55.283,374.684,-24.261,21.467,-42.212
C06085=1017.936,55.617,374.655,-24.262,21.467,-42.209
C06086=1017.932,55.953,374.626,-24.262,21.467,-42.205
C06087=1017.928,56.288,374.597,-24.263,21.466,-42.201
C06088=1017.924,56.622,374.568,-24.263,21.466,-42.197
C06089=1017.919,56.958,374.538,-24.264,21.466,-42.194
C06090=1017.915,57.293,374.510,-24.264,21.465,-42.192
C06091=1017.911,57.627,374.480,-24.264,21.465,-42.188
C06092=1017.907,57.963,374.451,-24.265,21.464,-42.184
C06093=1017.902,58.297,374.421,-24.266,21.465,-42.181
C06094=1017.898,58.633,374.393,-24.266,21.464,-42.177
C06095=1017.894,58.968,374.364,-24.267,21.464,-42.173
C06096=1017.889,59.303,374.334,-24.267,21.464,-42.170
C06097=1017.885,59.638,374.305,-24.268,21.464,-42.166
C06098=1017.881,59.973,374.276,-24.268,21.463,-42.163
C06099=1017.876,60.308,374.246,-24.268,21.462,-42.160
C06100=1017.873,60.643,374.217,-24.269,21.462,-42.157
C06101=1017.868,60.977,374.188,-24.269,21.462,-42.153
C06102=1017.864,61.313,374.158,-24.270,21.461,-42.149
C06103=1017.859,61.648,374.130,-24.270,21.462,-42.146
C06104=1017.855,61.983,374.100,-24.271,21.461,-42.142
C06105=1017.850,62.318,374.071,-24.271,21.461,-42.139
C06106=1017.846,62.654,374.041,-24.272,21.460,-42.135
C06107=1017.841,63.050,374.008,-24.272,21.460,-42.131
C06108=1017.838,63.274,373.987,-24.273,21.461,-42.130
C06109=1017.836,63.492,373.968,-24.273,21.460,-42.128
C06110=1017.834,63.866,373.933,-24.274,21.460,-42.124
C06111=1017.833,64.222,373.899,-24.274,21.459,-42.120
C06112=1017.833,64.608,373.863,-24.274,21.459,-42.116
C06113=1017.831,65.004,373.826,-24.275,21.458,-42.113
C06114=1017.830,65.380,373.790,-24.276,21.459,-42.108
C06115=1017.830,65.735,373.757,-24.276,21.457,-42.105
C06116=1017.828,66.074,373.725,-24.277,21.458,-42.102
C06117=1017.827,66.407,373.694,-24.277,21.457,-42.098
C06118=1017.827,66.742,373.662,-24.278,21.457,-42.094
C06119=1017.826,67.079,373.630,-24.278,21.457,-42.091
C06120=1017.825,67.416,373.598,-24.279,21.457,-42.087
C06121=1017.823,67.755,373.566,-24.279,21.456,-42.085
C06122=1017.823,68.094,373.534,-24.279,21.456,-42.082
C06123=1017.822,68.434,373.502,-24.280,21.456,-42.078
C06124=1017.820,68.775,373.470,-24.280,21.455,-42.074
C06125=1017.819,69.118,373.437,-24.281,21.456,-42.071
C06126=1017.819,69.462,373.405,-24.281,21.455,-42.067
C06127=1017.818,69.805,373.372,-24.282,21.455,-42.063
C06128=1017.816,70.149,373.339,-24.282,21.454,-42.061
C06129=1017.815,70.494,373.307,-24.283,21.454,-42.058
C06130=1017.814,70.838,373.275,-24.283,21.453,-42.054
C06131=1017.813,71.183,373.242,-24.284,21.454,-42.051
C06132=1017.812,71.527,373.209,-24.284,21.453,-42.047
C06133=1017.811,71.872,373.176,-24.285,21.453,-42.043
C06134=1017.810,72.217,373.144,-24.285,21.453,-42.041
C06135=1017.809,72.564,373.110,-24.285,21.452,-42.037
C06136=1017.809,72.912,373.078,-24.286,21.452,-42.034
C06137=1017.807,73.262,373.045,-24.286,21.451,-42.030
C06138=1017.806,73.613,373.011,-24.287,21.452,-42.027
C06139=1017.805,73.967,372.978,-24.288,21.451,-42.023
C06140=1017.804,74.322,372.944,-24.288,21.451,-42.019
C06141=1017.802,74.678,372.910,-24.288,21.451,-42.017
C06142=1017.802,75.036,372.875,-24.289,21.450,-42.013
C06143=1017.801,75.393,372.841,-24.289,21.450,-42.010
C06144=1017.799,75.748,372.807,-24.290,21.450,-42.006
C06145=1017.798,76.097,372.774,-24.290,21.449,-42.004
C06146=1017.798,76.439,372.741,-24.291,21.449,-42.001
C06147=1017.796,76.775,372.709,-24.291,21.449,-41.997
C06148=1017.795,77.105,372.678,-24.292,21.449,-41.994
C06149=1017.794,77.431,372.646,-24.292,21.449,-41.990
C06150=1017.793,77.755,372.616,-24.292,21.448,-41.987
C06151=1017.792,78.079,372.584,-24.293,21.448,-41.984
C06152=1017.792,78.403,372.553,-24.293,21.448,-41.980
C06153=1017.790,78.731,372.522,-24.294,21.447,-41.977
C06154=1017.789,79.063,372.490,-24.295,21.448,-41.973
C06155=1017.789,79.403,372.457,-24.295,21.446,-41.971
C06156=1017.787,79.748,372.424,-24.295,21.447,-41.968
C06157=1017.786,80.098,372.391,-24.296,21.446,-41.964
C06158=1017.785,80.454,372.357,-24.296,21.446,-41.962
C06159=1017.783,80.810,372.322,-24.297,21.446,-41.958
C06160=1017.783,81.167,372.288,-24.297,21.445,-41.955
C06161=1017.781,81.523,372.254,-24.298,21.446,-41.951
C06162=1017.780,81.878,372.220,-24.298,21.445,-41.947
C06163=1017.779,82.232,372.186,-24.298,21.444,-41.945
C06164=1017.778,82.586,372.151,-24.299,21.444,-41.942
C06165=1017.776,82.940,372.117,-24.299,21.444,-41.938
C06166=1017.775,83.292,372.084,-24.300,21.444,-41.935
C06167=1017.774,83.642,372.050,-24.300,21.444,-41.931
C06168=1017.773,83.992,372.016,-24.301,21.443,-41.929
C06169=1017.772,84.341,371.982,-24.301,21.443,-41.925
C06170=1017.770,84.689,371.949,-24.302,21.443,-41.922
C06171=1017.770,85.036,371.915,-24.302,21.443,-41.918
C06172=1017.768,85.381,371.882,-24.302,21.442,-41.916
C06173=1017.768,85.725,371.848,-24.303,21.442,-41.912
C06174=1017.766,86.068,371.815,-24.303,21.442,-41.909
C06175=1017.766,86.410,371.782,-24.304,21.441,-41.906
C06176=1017.764,86.751,371.750,-24.304,21.441,-41.903
C06177=1017.763,87.090,371.717,-24.305,21.441,-41.899
C06178=1017.762,87.427,371.684,-24.305,21.441,-41.898
C06179=1017.761,87.760,371.652,-24.305,21.440,-41.894
C06180=1017.760,88.086,371.621,-24.306,21.441,-41.890
C06181=1017.759,88.408,371.589,-24.306,21.439,-41.888
C06182=1017.757,88.729,371.558,-24.307,21.440,-41.885
C06183=1017.756,89.050,371.527,-24.307,21.439,-41.881
C06184=1017.755,89.374,371.495,-24.308,21.439,-41.879
C06185=1017.755,89.704,371.463,-24.308,21.440,-41.876
C06186=1017.752,90.037,371.431,-24.308,21.438,-41.874
C06187=1017.752,90.371,371.399,-24.309,21.439,-41.870
C06188=1017.751,90.706,371.366,-24.309,21.438,-41.866
C06189=1017.750,91.040,371.333,-24.310,21.438,-41.865
C06190=1017.748,91.374,371.301,-24.310,21.438,-41.861
C06191=1017.747,91.709,371.268,-24.311,21.438,-41.857
C06192=1017.747,92.044,371.236,-24.311,21.437,-41.855
C06193=1017.745,92.378,371.203,-24.311,21.437,-41.852
C06194=1017.744,92.712,371.171,-24.312,21.436,-41.849
C06195=1017.742,93.047,371.138,-24.312,21.437,-41.846
C06196=1017.741,93.382,371.105,-24.313,21.436,-41.842
C06197=1017.741,93.715,371.073,-24.313,21.436,-41.841
C06198=1017.739,94.049,371.040,-24.314,21.436,-41.837
C06199=1017.738,94.384,371.008,-24.314,21.436,-41.833
C06200=1017.737,94.719,370.975,-24.314,21.436,-41.832
C06201=1017.735,95.053,370.942,-24.315,21.435,-41.828
C06202=1017.734,95.387,370.909,-24.315,21.435,-41.826
C06203=1017.733,95.721,370.877,-24.316,21.435,-41.822
C06204=1017.732,96.055,370.845,-24.316,21.435,-41.819
C06205=1017.731,96.390,370.812,-24.316,21.434,-41.817
C06206=1017.730,96.724,370.779,-24.317,21.434,-41.813
C06207=1017.728,97.058,370.746,-24.317,21.434,-41.811
C06208=1017.727,97.393,370.714,-24.318,21.434,-41.808
C06209=1017.726,97.726,370.680,-24.318,21.433,-41.806
C06210=1017.724,98.061,370.648,-24.318,21.433,-41.802
C06211=1017.723,98.396,370.615,-24.319,21.433,-41.799
C06212=1017.723,98.729,370.582,-24.319,21.432,-41.796
C06213=1017.722,99.064,370.550,-24.320,21.433,-41.793
C06214=1017.720,99.397,370.517,-24.320,21.432,-41.791
C06215=1017.719,99.732,370.484,-24.320,21.432,-41.787
C06216=1017.717,100.066,370.452,-24.321,21.432,-41.785
C06217=1017.716,100.400,370.419,-24.321,21.431,-41.782
C06218=1017.715,100.735,370.386,-24.322,21.432,-41.778
C06219=1017.714,101.069,370.352,-24.322,21.431,-41.776
C06220=1017.713,101.403,370.320,-24.323,21.431,-41.773
C06221=1017.711,101.737,370.287,-24.323,21.431,-41.771
C06222=1017.710,102.071,370.254,-24.323,21.430,-41.767
C06223=1017.709,102.405,370.221,-24.324,21.430,-41.765
C06224=1017.707,102.739,370.188,-24.324,21.431,-41.762
C06225=1017.707,103.073,370.155,-24.324,21.429,-41.760
C06226=1017.705,103.408,370.122,-24.325,21.430,-41.756
C06227=1017.704,103.741,370.089,-24.325,21.429,-41.752
C06228=1017.703,104.075,370.056,-24.326,21.429,-41.751
C06229=1017.701,104.410,370.023,-24.326,21.430,-41.747
C06230=1017.700,104.743,369.990,-24.326,21.428,-41.745
C06231=1017.699,105.078,369.958,-24.327,21.429,-41.742
C06232=1017.698,105.411,369.924,-24.327,21.428,-41.739
C06233=1017.697,105.746,369.891,-24.328,21.428,-41.736
C06234=1017.696,106.080,369.858,-24.328,21.428,-41.734
C06235=1017.694,106.414,369.825,-24.328,21.427,-41.730
C06236=1017.693,106.748,369.792,-24.329,21.427,-41.728
C06237=1017.692,107.082,369.759,-24.329,21.428,-41.725
C06238=1017.690,107.416,369.726,-24.329,21.427,-41.723
C06239=1017.689,107.749,369.693,-24.330,21.427,-41.719
C06240=1017.688,108.083,369.660,-24.330,21.427,-41.718
C06241=1017.687,108.418,369.627,-24.331,21.426,-41.714
C06242=1017.686,108.752,369.594,-24.331,21.426,-41.712
C06243=1017.685,109.086,369.560,-24.332,21.426,-41.708
C06244=1017.683,109.420,369.528,-24.332,21.425,-41.706
C06245=1017.681,109.754,369.494,-24.332,21.426,-41.703
C06246=1017.680,110.088,369.461,-24.333,21.425,-41.701
C06247=1017.679,110.421,369.428,-24.333,21.425,-41.697
C06248=1017.678,110.755,369.395,-24.333,21.425,-41.695
C06249=1017.677,111.090,369.362,-24.334,21.424,-41.692
C06250=1017.676,111.424,369.328,-24.334,21.424,-41.690
C06251=1017.675,111.758,369.295,-24.335,21.425,-41.686
C06252=1017.674,112.091,369.262,-24.335,21.423,-41.684
C06253=1017.672,112.425,369.228,-24.335,21.424,-41.681
C06254=1017.670,112.759,369.195,-24.336,21.424,-41.679
C06255=1017.669,113.093,369.162,-24.336,21.423,-41.675
C06256=1017.668,113.427,369.129,-24.336,21.423,-41.673
C06257=1017.667,113.762,369.096,-24.337,21.423,-41.670
C06258=1017.665,114.096,369.062,-24.337,21.422,-41.668
C06259=1017.664,114.429,369.029,-24.338,21.423,-41.664
C06260=1017.663,114.763,368.995,-24.338,21.422,-41.662
C06261=1017.662,115.097,368.962,-24.338,21.421,-41.660
C06262=1017.661,115.430,368.929,-24.339,21.422,-41.657
C06263=1017.659,115.764,368.895,-24.339,21.422,-41.655
C06264=1017.658,116.099,368.862,-24.340,21.422,-41.652
C06265=1017.657,116.433,368.828,-24.340,21.421,-41.649
C06266=1017.656,116.766,368.795,-24.340,21.421,-41.646
C06267=1017.654,117.100,368.761,-24.341,21.421,-41.644
C06268=1017.653,117.434,368.728,-24.341,21.421,-41.640
C06269=1017.652,117.769,368.695,-24.341,21.420,-41.638
C06270=1017.651,118.103,368.662,-24.342,21.421,-41.635
C06271=1017.649,118.437,368.628,-24.342,21.420,-41.633
C06272=1017.647,118.771,368.595,-24.342,21.419,-41.631
C06273=1017.646,119.104,368.562,-24.343,21.420,-41.628
C06274=1017.645,119.438,368.527,-24.343,21.419,-41.625
C06275=1017.644,119.772,368.494,-24.344,21.419,-41.622
C06276=1017.643,120.106,368.460,-24.344,21.419,-41.620
C06277=1017.641,120.440,368.427,-24.345,21.419,-41.617
C06278=1017.640,120.774,368.393,-24.345,21.418,-41.614
C06279=1017.639,121.108,368.360,-24.345,21.418,-41.613
C06280=1017.637,121.442,368.326,-24.346,21.418,-41.609
C06281=1017.636,121.776,368.293,-24.346,21.417,-41.607
C06282=1017.634,122.110,368.259,-24.346,21.418,-41.604
C06283=1017.633,122.444,368.226,-24.347,21.418,-41.602
C06284=1017.632,122.778,368.192,-24.347,21.418,-41.598
C06285=1017.631,123.112,368.158,-24.347,21.417,-41.596
C06286=1017.629,123.446,368.125,-24.348,21.417,-41.594
C06287=1017.628,123.780,368.090,-24.348,21.417,-41.591
C06288=1017.627,124.114,368.057,-24.348,21.417,-41.589
C06289=1017.626,124.447,368.024,-24.349,21.416,-41.585
C06290=1017.624,124.781,367.990,-24.349,21.416,-41.583
C06291=1017.624,125.116,367.956,-24.349,21.416,-41.581
C06292=1017.622,125.450,367.923,-24.350,21.416,-41.578
C06293=1017.620,125.784,367.889,-24.350,21.415,-41.576
C06294=1017.619,126.118,367.854,-24.351,21.416,-41.572
C06295=1017.618,126.451,367.821,-24.351,21.415,-41.571
C06296=1017.616,126.785,367.787,-24.351,21.415,-41.569
C06297=1017.616,127.120,367.754,-24.352,21.415,-41.565
C06298=1017.614,127.454,367.720,-24.352,21.415,-41.563
C06299=1017.613,127.788,367.687,-24.352,21.414,-41.561
C06300=1017.612,128.122,367.652,-24.353,21.415,-41.558
C06301=1017.610,128.455,367.619,-24.353,21.414,-41.555
C06302=1017.609,128.789,367.585,-24.354,21.414,-41.552
C06303=1017.607,129.124,367.551,-24.354,21.414,-41.550
C06304=1017.606,129.458,367.517,-24.354,21.414,-41.548
C06305=1017.605,129.792,367.483,-24.355,21.413,-41.545
C06306=1017.604,130.126,367.449,-24.355,21.413,-41.543
C06307=1017.602,130.460,367.415,-24.355,21.413,-41.541
C06308=1017.601,130.794,367.382,-24.356,21.413,-41.538
C06309=1017.600,131.128,367.347,-24.356,21.412,-41.535
C06310=1017.598,131.462,367.313,-24.356,21.412,-41.532
C06311=1017.597,131.796,367.280,-24.357,21.412,-41.530
C06312=1017.596,132.131,367.246,-24.357,21.412,-41.528
C06313=1017.594,132.464,367.211,-24.357,21.412,-41.525
C06314=1017.594,132.799,367.178,-24.358,21.411,-41.523
C06315=1017.592,133.133,367.144,-24.358,21.411,-41.521
C06316=1017.591,133.467,367.109,-24.358,21.411,-41.517
C06317=1017.590,133.801,367.076,-24.359,21.411,-41.515
C06318=1017.588,134.135,367.042,-24.359,21.410,-41.513
C06319=1017.586,134.469,367.008,-24.359,21.411,-41.510
C06320=1017.585,134.803,366.973,-24.360,21.410,-41.508
C06321=1017.584,135.137,366.940,-24.360,21.410,-41.506
C06322=1017.583,135.471,366.905,-24.361,21.411,-41.503
C06323=1017.581,135.794,366.873,-24.361,21.410,-41.501
C06324=1017.581,136.095,366.842,-24.361,21.410,-41.499
C06325=1017.579,136.373,366.814,-24.361,21.410,-41.497
C06326=1017.578,136.638,366.786,-24.361,21.409,-41.495
C06327=1017.577,136.903,366.759,-24.362,21.409,-41.491
C06328=1017.576,137.179,366.731,-24.362,21.409,-41.490
C06329=1017.576,137.476,366.701,-24.363,21.409,-41.488
C06330=1017.574,137.798,366.667,-24.363,21.408,-41.486
C06331=1017.573,138.139,366.632,-24.363,21.408,-41.484
C06332=1017.571,138.495,366.597,-24.364,21.408,-41.480
C06333=1017.570,138.907,366.554,-24.364,21.408,-41.477
C06334=1017.569,139.135,366.531,-24.364,21.408,-41.475
C06335=1017.567,139.372,366.507,-24.365,21.408,-41.473
C06336=1017.567,139.614,366.482,-24.365,21.408,-41.473
C06337=1017.566,139.855,366.457,-24.365,21.408,-41.471
C06338=1017.566,140.088,366.433,-24.365,21.408,-41.470
C06339=1017.564,140.308,366.411,-24.365,21.407,-41.469
C06340=1017.563,140.701,366.371,-24.366,21.407,-41.465
C06341=1017.562,141.046,366.335,-24.366,21.407,-41.462
C06342=1017.560,141.385,366.300,-24.367,21.407,-41.460
C06343=1017.559,141.725,366.265,-24.367,21.407,-41.457
C06344=1017.558,142.065,366.230,-24.367,21.406,-41.455
C06345=1017.555,142.406,366.195,-24.368,21.406,-41.453
C06346=1017.555,142.748,366.160,-24.368,21.407,-41.449
C06347=1017.554,143.089,366.125,-24.368,21.406,-41.448
C06348=1017.552,143.432,366.090,-24.369,21.405,-41.445
C06349=1017.551,143.774,366.055,-24.369,21.406,-41.442
C06350=1017.549,144.119,366.019,-24.369,21.405,-41.440
C06351=1017.548,144.463,365.984,-24.370,21.405,-41.438
C06352=1017.547,144.807,365.948,-24.370,21.406,-41.435
C06353=1017.546,145.152,365.912,-24.370,21.405,-41.432
C06354=1017.544,145.498,365.877,-24.371,21.404,-41.431
C06355=1017.543,145.843,365.842,-24.371,21.405,-41.427
C06356=1017.542,146.189,365.806,-24.371,21.405,-41.425
C06357=1017.540,146.535,365.770,-24.372,21.404,-41.424
C06358=1017.535,146.882,365.737,-24.372,21.404,-41.420
C06359=1017.517,147.227,365.712,-24.372,21.404,-41.418
C06360=1017.901,147.255,365.472,-24.372,21.404,-41.418
C06361=1017.920,146.909,365.497,-24.372,21.404,-41.420
C06362=1017.926,146.563,365.530,-24.372,21.404,-41.424
C06363=1017.928,146.217,365.566,-24.371,21.405,-41.425
C06364=1017.928,145.871,365.601,-24.371,21.405,-41.427
C06365=1017.930,145.525,365.637,-24.371,21.404,-41.431
C06366=1017.932,145.180,365.672,-24.370,21.405,-41.432
C06367=1017.933,144.835,365.708,-24.370,21.406,-41.435
C06368=1017.934,144.491,365.744,-24.370,21.405,-41.438
C06369=1017.935,144.146,365.779,-24.369,21.405,-41.440
C06370=1017.937,143.803,365.814,-24.369,21.406,-41.442
C06371=1017.938,143.459,365.849,-24.369,21.405,-41.445
C06372=1017.939,143.117,365.884,-24.368,21.406,-41.448
C06373=1017.941,142.775,365.919,-24.368,21.407,-41.449
C06374=1017.942,142.434,365.955,-24.368,21.406,-41.453
C06375=1017.943,142.093,365.990,-24.367,21.406,-41.455
C06376=1017.944,141.753,366.025,-24.367,21.407,-41.457
C06377=1017.946,141.413,366.059,-24.367,21.407,-41.460
C06378=1017.947,141.074,366.094,-24.366,21.407,-41.462
C06379=1017.948,140.729,366.130,-24.366,21.407,-41.465
C06380=1017.950,140.336,366.170,-24.365,21.407,-41.469
C06381=1017.951,140.116,366.193,-24.365,21.408,-41.470
C06382=1017.951,139.883,366.217,-24.365,21.408,-41.471
C06383=1017.952,139.642,366.241,-24.365,21.408,-41.473
C06384=1017.953,139.400,366.266,-24.365,21.408,-41.473
C06385=1017.954,139.162,366.290,-24.364,21.408,-41.475
C06386=1017.955,138.935,366.314,-24.364,21.408,-41.477
C06387=1017.956,138.523,366.356,-24.364,21.408,-41.480
C06388=1017.958,138.167,366.392,-24.363,21.408,-41.484
C06389=1017.959,137.826,366.427,-24.363,21.408,-41.486
C06390=1017.961,137.504,366.460,-24.363,21.409,-41.488
C06391=1017.962,137.207,366.491,-24.362,21.409,-41.490
C06392=1017.963,136.931,366.519,-24.362,21.409,-41.491
C06393=1017.963,136.666,366.546,-24.361,21.409,-41.495
C06394=1017.965,136.401,366.573,-24.361,21.410,-41.497
C06395=1017.966,136.123,366.602,-24.361,21.410,-41.499
C06396=1017.967,135.822,366.632,-24.361,21.410,-41.501
C06397=1017.968,135.499,366.665,-24.361,21.411,-41.503
C06398=1017.970,135.165,366.699,-24.360,21.410,-41.506
C06399=1017.972,134.831,366.733,-24.360,21.410,-41.508
C06400=1017.972,134.497,366.767,-24.359,21.411,-41.510
C06401=1017.974,134.163,366.801,-24.359,21.410,-41.513
C06402=1017.975,133.829,366.835,-24.359,21.411,-41.515
C06403=1017.976,133.495,366.869,-24.358,21.411,-41.517
C06404=1017.977,133.161,366.903,-24.358,21.411,-41.521
C06405=1017.979,132.826,366.938,-24.358,21.411,-41.523
C06406=1017.980,132.492,366.971,-24.357,21.412,-41.525
C06407=1017.981,132.158,367.006,-24.357,21.412,-41.528
C06408=1017.983,131.824,367.040,-24.357,21.412,-41.530
C06409=1017.984,131.490,367.073,-24.356,21.412,-41.532
C06410=1017.985,131.156,367.107,-24.356,21.412,-41.535
C06411=1017.987,130.822,367.141,-24.356,21.413,-41.538
C06412=1017.987,130.488,367.175,-24.355,21.413,-41.541
C06413=1017.989,130.154,367.209,-24.355,21.413,-41.543
C06414=1017.990,129.819,367.242,-24.355,21.413,-41.545
C06415=1017.991,129.486,367.277,-24.354,21.414,-41.548
C06416=1017.993,129.152,367.311,-24.354,21.414,-41.550
C06417=1017.994,128.817,367.344,-24.354,21.414,-41.552
C06418=1017.996,128.483,367.378,-24.353,21.414,-41.555
C06419=1017.996,128.150,367.412,-24.353,21.415,-41.558
C06420=1017.998,127.816,367.446,-24.352,21.414,-41.561
C06421=1017.999,127.482,367.480,-24.352,21.415,-41.563
C06422=1018.001,127.147,367.514,-24.352,21.415,-41.565
C06423=1018.002,126.813,367.547,-24.351,21.415,-41.569
C06424=1018.003,126.480,367.581,-24.351,21.415,-41.571
C06425=1018.004,126.146,367.615,-24.351,21.416,-41.572
C06426=1018.006,125.812,367.649,-24.350,21.415,-41.576
C06427=1018.007,125.478,367.682,-24.350,21.416,-41.578
C06428=1018.008,125.143,367.716,-24.349,21.416,-41.581
C06429=1018.009,124.809,367.749,-24.349,21.416,-41.583
C06430=1018.011,124.475,367.783,-24.349,21.416,-41.585
C06431=1018.012,124.142,367.818,-24.348,21.417,-41.589
C06432=1018.013,123.808,367.851,-24.348,21.417,-41.591
C06433=1018.015,123.474,367.885,-24.348,21.417,-41.594
C06434=1018.016,123.140,367.918,-24.347,21.417,-41.596
C06435=1018.017,122.805,367.952,-24.347,21.418,-41.598
C06436=1018.018,122.472,367.985,-24.347,21.418,-41.602
C06437=1018.020,122.138,368.018,-24.346,21.418,-41.604
C06438=1018.022,121.804,368.052,-24.346,21.417,-41.607
C06439=1018.022,121.470,368.087,-24.346,21.418,-41.609
C06440=1018.024,121.136,368.120,-24.345,21.418,-41.613
C06441=1018.025,120.802,368.154,-24.345,21.418,-41.614
C06442=1018.026,120.469,368.187,-24.345,21.419,-41.617
C06443=1018.027,120.134,368.221,-24.344,21.419,-41.620
C06444=1018.029,119.800,368.254,-24.344,21.419,-41.622
C06445=1018.030,119.466,368.287,-24.343,21.419,-41.625
C06446=1018.032,119.132,368.321,-24.343,21.420,-41.628
C06447=1018.032,118.798,368.355,-24.342,21.419,-41.631
C06448=1018.033,118.464,368.388,-24.342,21.420,-41.633
C06449=1018.035,118.130,368.421,-24.342,21.421,-41.635
C06450=1018.037,117.796,368.455,-24.341,21.420,-41.638
C06451=1018.038,117.463,368.488,-24.341,21.421,-41.640
C06452=1018.039,117.129,368.522,-24.341,21.421,-41.644
C06453=1018.040,116.794,368.556,-24.340,21.421,-41.646
C06454=1018.041,116.461,368.589,-24.340,21.421,-41.649
C06455=1018.043,116.127,368.622,-24.340,21.422,-41.652
C06456=1018.044,115.793,368.655,-24.339,21.422,-41.655
C06457=1018.046,115.459,368.689,-24.339,21.422,-41.657
C06458=1018.047,115.125,368.722,-24.338,21.421,-41.660
C06459=1018.047,114.791,368.756,-24.338,21.422,-41.662
C06460=1018.049,114.457,368.789,-24.338,21.423,-41.664
C06461=1018.050,114.123,368.822,-24.337,21.422,-41.668
C06462=1018.052,113.789,368.856,-24.337,21.423,-41.670
C06463=1018.053,113.455,368.889,-24.336,21.423,-41.673
C06464=1018.054,113.121,368.922,-24.336,21.423,-41.675
C06465=1018.055,112.787,368.956,-24.336,21.424,-41.679
C06466=1018.056,112.453,368.989,-24.335,21.424,-41.681
C06467=1018.057,112.120,369.022,-24.335,21.423,-41.684
C06468=1018.059,111.785,369.056,-24.335,21.425,-41.686
C06469=1018.061,111.451,369.088,-24.334,21.424,-41.690
C06470=1018.062,111.117,369.122,-24.334,21.424,-41.692
C06471=1018.063,110.784,369.155,-24.333,21.425,-41.695
C06472=1018.064,110.449,369.188,-24.333,21.425,-41.697
C06473=1018.065,110.116,369.222,-24.333,21.425,-41.701
C06474=1018.066,109.781,369.254,-24.332,21.426,-41.703
C06475=1018.067,109.447,369.287,-24.332,21.425,-41.706
C06476=1018.069,109.114,369.321,-24.332,21.426,-41.708
C06477=1018.071,108.780,369.354,-24.331,21.426,-41.712
C06478=1018.072,108.445,369.387,-24.331,21.426,-41.714
C06479=1018.073,108.112,369.420,-24.330,21.427,-41.718
C06480=1018.074,107.777,369.454,-24.330,21.427,-41.719
C06481=1018.075,107.444,369.487,-24.329,21.427,-41.723
C06482=1018.076,107.109,369.519,-24.329,21.428,-41.725
C06483=1018.078,106.775,369.553,-24.329,21.427,-41.728
C06484=1018.079,106.442,369.586,-24.328,21.427,-41.730
C06485=1018.080,106.107,369.618,-24.328,21.428,-41.734
C06486=1018.081,105.774,369.652,-24.328,21.428,-41.736
C06487=1018.083,105.440,369.685,-24.327,21.428,-41.739
C06488=1018.084,105.105,369.718,-24.327,21.429,-41.742
C06489=1018.085,104.771,369.751,-24.326,21.428,-41.745
C06490=1018.086,104.437,369.783,-24.326,21.430,-41.747
C06491=1018.087,104.103,369.817,-24.326,21.429,-41.751
C06492=1018.089,103.769,369.850,-24.325,21.429,-41.752
C06493=1018.090,103.435,369.882,-24.325,21.430,-41.756
C06494=1018.091,103.101,369.915,-24.324,21.429,-41.760
C06495=1018.092,102.766,369.948,-24.324,21.431,-41.762
C06496=1018.093,102.433,369.982,-24.324,21.430,-41.765
C06497=1018.095,102.098,370.014,-24.323,21.430,-41.767
C06498=1018.096,101.764,370.047,-24.323,21.431,-41.771
C06499=1018.097,101.430,370.080,-24.323,21.431,-41.773
C06500=1018.099,101.096,370.113,-24.322,21.431,-41.776
C06501=1018.100,100.762,370.146,-24.322,21.432,-41.778
C06502=1018.101,100.428,370.179,-24.321,21.431,-41.782
C06503=1018.102,100.093,370.212,-24.321,21.432,-41.785
C06504=1018.103,99.760,370.245,-24.320,21.432,-41.787
C06505=1018.104,99.426,370.277,-24.320,21.432,-41.791
C06506=1018.105,99.092,370.310,-24.320,21.433,-41.793
C06507=1018.107,98.757,370.342,-24.319,21.432,-41.796
C06508=1018.108,98.422,370.375,-24.319,21.433,-41.799
C06509=1018.109,98.089,370.409,-24.318,21.433,-41.802
C06510=1018.110,97.754,370.441,-24.318,21.433,-41.806
C06511=1018.112,97.420,370.474,-24.318,21.434,-41.808
C06512=1018.113,97.086,370.507,-24.317,21.434,-41.811
C06513=1018.114,96.752,370.539,-24.317,21.434,-41.813
C06514=1018.115,96.417,370.572,-24.316,21.434,-41.817
C06515=1018.116,96.083,370.605,-24.316,21.435,-41.819
C06516=1018.117,95.749,370.637,-24.316,21.435,-41.822
C06517=1018.119,95.415,370.670,-24.315,21.435,-41.826
C06518=1018.120,95.081,370.703,-24.315,21.435,-41.828
C06519=1018.121,94.746,370.736,-24.314,21.436,-41.832
C06520=1018.122,94.412,370.768,-24.314,21.436,-41.833
C06521=1018.123,94.078,370.800,-24.314,21.436,-41.837
C06522=1018.125,93.743,370.833,-24.313,21.436,-41.841
C06523=1018.125,93.409,370.866,-24.313,21.436,-41.842
C06524=1018.127,93.075,370.899,-24.312,21.437,-41.846
C06525=1018.128,92.740,370.931,-24.312,21.436,-41.849
C06526=1018.129,92.406,370.963,-24.311,21.437,-41.852
C06527=1018.130,92.071,370.996,-24.311,21.437,-41.855
C06528=1018.131,91.737,371.029,-24.311,21.438,-41.857
C06529=1018.133,91.402,371.061,-24.310,21.438,-41.861
C06530=1018.134,91.068,371.094,-24.310,21.438,-41.865
C06531=1018.134,90.733,371.126,-24.309,21.438,-41.866
C06532=1018.136,90.399,371.158,-24.309,21.439,-41.870
C06533=1018.137,90.065,371.192,-24.308,21.438,-41.874
C06534=1018.138,89.731,371.224,-24.308,21.440,-41.876
C06535=1018.139,89.402,371.256,-24.308,21.439,-41.879
C06536=1018.140,89.078,371.287,-24.307,21.439,-41.881
C06537=1018.142,88.757,371.318,-24.307,21.440,-41.885
C06538=1018.142,88.436,371.349,-24.306,21.439,-41.888
C06539=1018.143,88.114,371.381,-24.306,21.441,-41.890
C06540=1018.144,87.787,371.412,-24.305,21.440,-41.894
C06541=1018.146,87.455,371.444,-24.305,21.441,-41.898
C06542=1018.147,87.118,371.477,-24.305,21.441,-41.899
C06543=1018.147,86.778,371.510,-24.304,21.441,-41.903
C06544=1018.149,86.438,371.542,-24.304,21.441,-41.906
C06545=1018.151,86.096,371.576,-24.303,21.442,-41.909
C06546=1018.152,85.752,371.609,-24.303,21.442,-41.912
C06547=1018.153,85.409,371.643,-24.302,21.442,-41.916
C06548=1018.154,85.063,371.676,-24.302,21.443,-41.918
C06549=1018.155,84.717,371.710,-24.302,21.443,-41.922
C06550=1018.156,84.369,371.743,-24.301,21.443,-41.925
C06551=1018.158,84.020,371.777,-24.301,21.443,-41.929
C06552=1018.158,83.670,371.810,-24.300,21.444,-41.931
C06553=1018.159,83.319,371.845,-24.300,21.444,-41.935
C06554=1018.160,82.967,371.878,-24.299,21.444,-41.938
C06555=1018.161,82.614,371.912,-24.299,21.444,-41.942
C06556=1018.163,82.260,371.946,-24.298,21.444,-41.945
C06557=1018.163,81.906,371.980,-24.298,21.445,-41.947
C06558=1018.166,81.550,372.015,-24.298,21.446,-41.951
C06559=1018.166,81.195,372.048,-24.297,21.445,-41.955
C06560=1018.168,80.838,372.083,-24.297,21.446,-41.958
C06561=1018.168,80.481,372.118,-24.296,21.446,-41.962
C06562=1018.170,80.127,372.151,-24.296,21.446,-41.964
C06563=1018.171,79.775,372.185,-24.295,21.447,-41.968
C06564=1018.172,79.430,372.218,-24.295,21.446,-41.971
C06565=1018.173,79.092,372.251,-24.295,21.448,-41.973
C06566=1018.174,78.759,372.282,-24.294,21.447,-41.977
C06567=1018.175,78.431,372.314,-24.293,21.448,-41.980
C06568=1018.176,78.106,372.345,-24.293,21.448,-41.984
C06569=1018.177,77.783,372.376,-24.292,21.448,-41.987
C06570=1018.178,77.458,372.407,-24.292,21.449,-41.990
C06571=1018.179,77.133,372.438,-24.292,21.449,-41.994
C06572=1018.180,76.802,372.470,-24.291,21.449,-41.997
C06573=1018.181,76.466,372.502,-24.291,21.449,-42.001
C06574=1018.182,76.124,372.535,-24.290,21.449,-42.004
C06575=1018.183,75.775,372.568,-24.290,21.450,-42.006
C06576=1018.184,75.422,372.601,-24.289,21.450,-42.010
C06577=1018.186,75.064,372.635,-24.289,21.450,-42.013
C06578=1018.186,74.707,372.670,-24.288,21.451,-42.017
C06579=1018.187,74.350,372.704,-24.288,21.451,-42.019
C06580=1018.188,73.994,372.738,-24.288,21.451,-42.023
C06581=1018.190,73.641,372.772,-24.287,21.452,-42.027
C06582=1018.190,73.289,372.805,-24.286,21.451,-42.030
C06583=1018.192,72.940,372.838,-24.286,21.452,-42.034
C06584=1018.193,72.592,372.871,-24.285,21.452,-42.037
C06585=1018.194,72.246,372.904,-24.285,21.453,-42.041
C06586=1018.195,71.899,372.937,-24.285,21.453,-42.043
C06587=1018.196,71.555,372.970,-24.284,21.453,-42.047
C06588=1018.197,71.210,373.003,-24.284,21.454,-42.051
C06589=1018.198,70.866,373.035,-24.283,21.453,-42.054
C06590=1018.199,70.522,373.068,-24.283,21.454,-42.058
C06591=1018.201,70.178,373.101,-24.282,21.454,-42.061
C06592=1018.201,69.833,373.133,-24.282,21.455,-42.063
C06593=1018.202,69.489,373.166,-24.281,21.455,-42.067
C06594=1018.203,69.145,373.198,-24.281,21.456,-42.071
C06595=1018.204,68.803,373.231,-24.280,21.455,-42.074
C06596=1018.205,68.462,373.263,-24.280,21.456,-42.078
C06597=1018.206,68.122,373.296,-24.279,21.456,-42.082
C06598=1018.207,67.783,373.327,-24.279,21.456,-42.085
C06599=1018.208,67.445,373.359,-24.279,21.457,-42.087
C06600=1018.209,67.107,373.391,-24.278,21.457,-42.091
C06601=1018.210,66.770,373.422,-24.278,21.457,-42.094
C06602=1018.211,66.435,373.454,-24.277,21.457,-42.098
C06603=1018.211,66.101,373.486,-24.277,21.458,-42.102
C06604=1018.213,65.762,373.518,-24.276,21.457,-42.105
C06605=1018.213,65.409,373.551,-24.276,21.459,-42.108
C06606=1018.214,65.031,373.587,-24.275,21.458,-42.113
C06607=1018.216,64.636,373.624,-24.274,21.459,-42.116
C06608=1018.217,64.249,373.661,-24.274,21.459,-42.120
C06609=1018.218,63.893,373.694,-24.274,21.460,-42.124
C06610=1018.219,63.520,373.729,-24.273,21.460,-42.128
C06611=1018.221,63.302,373.748,-24.273,21.461,-42.130
C06612=1018.224,63.078,373.769,-24.272,21.460,-42.131
C06613=1018.229,62.682,373.803,-24.272,21.460,-42.135
C06614=1018.233,62.346,373.832,-24.271,21.461,-42.139
C06615=1018.238,62.010,373.862,-24.271,21.461,-42.142
C06616=1018.242,61.676,373.891,-24.270,21.462,-42.146
C06617=1018.246,61.341,373.920,-24.270,21.461,-42.149
C06618=1018.250,61.005,373.950,-24.269,21.462,-42.153
C06619=1018.255,60.671,373.979,-24.269,21.462,-42.157
C06620=1018.258,60.336,374.008,-24.268,21.462,-42.160
C06621=1018.263,60.000,374.038,-24.268,21.463,-42.163
C06622=1018.268,59.665,374.066,-24.268,21.464,-42.166
C06623=1018.271,59.331,374.096,-24.267,21.464,-42.170
C06624=1018.276,58.995,374.126,-24.267,21.464,-42.173
C06625=1018.280,58.661,374.155,-24.266,21.464,-42.177
C06626=1018.284,58.325,374.184,-24.266,21.465,-42.181
C06627=1018.288,57.991,374.213,-24.265,21.464,-42.184
C06628=1018.293,57.655,374.242,-24.264,21.465,-42.188
C06629=1018.297,57.320,374.271,-24.264,21.465,-42.192
C06630=1018.300,56.985,374.301,-24.264,21.466,-42.194
C06631=1018.305,56.651,374.330,-24.263,21.466,-42.197
C06632=1018.308,56.316,374.359,-24.263,21.466,-42.201
C06633=1018.313,55.980,374.389,-24.262,21.467,-42.205
C06634=1018.317,55.645,374.418,-24.262,21.467,-42.209
C06635=1018.321,55.310,374.447,-24.261,21.467,-42.212
C06636=1018.325,54.975,374.476,-24.261,21.467,-42.216
C06637=1018.329,54.640,374.505,-24.260,21.468,-42.220
C06638=1018.333,54.305,374.534,-24.260,21.468,-42.223
C06639=1018.337,53.997,374.561,-24.259,21.468,-42.227
C06640=1018.341,53.635,374.592,-24.259,21.468,-42.230
C06641=1018.345,53.300,374.621,-24.258,21.469,-42.234
C06642=1018.348,52.965,374.651,-24.258,21.469,-42.238
C06643=1018.353,52.630,374.680,-24.257,21.470,-42.240
C06644=1018.356,52.295,374.709,-24.257,21.470,-42.244
C06645=1018.360,51.960,374.738,-24.256,21.470,-42.247
C06646=1018.364,51.625,374.767,-24.256,21.471,-42.251
C06647=1018.368,51.291,374.796,-24.255,21.471,-42.254
C06648=1018.372,50.955,374.825,-24.255,21.471,-42.258
C06649=1018.376,50.620,374.855,-24.254,21.471,-42.262
C06650=1018.380,50.285,374.884,-24.254,21.472,-42.266
C06651=1018.383,49.950,374.913,-24.253,21.472,-42.269
C06652=1018.387,49.616,374.941,-24.253,21.472,-42.273
C06653=1018.391,49.280,374.970,-24.252,21.473,-42.277
C06654=1018.395,48.945,375.000,-24.252,21.473,-42.280
C06655=1018.399,48.610,375.029,-24.251,21.473,-42.284
C06656=1018.402,48.275,375.058,-24.251,21.473,-42.287
C06657=1018.406,47.941,375.086,-24.250,21.474,-42.291
C06658=1018.410,47.605,375.115,-24.250,21.474,-42.295
C06659=1018.414,47.271,375.145,-24.249,21.475,-42.299
C06660=1018.417,46.935,375.173,-24.249,21.475,-42.302
C06661=1018.420,46.601,375.203,-24.248,21.475,-42.306
C06662=1018.425,46.266,375.231,-24.248,21.475,-42.309
C06663=1018.428,45.931,375.260,-24.247,21.476,-42.313
C06664=1018.432,45.596,375.289,-24.247,21.476,-42.317
C06665=1018.436,45.261,375.318,-24.246,21.477,-42.321
C06666=1018.438,44.926,375.347,-24.246,21.477,-42.325
C06667=1018.443,44.591,375.376,-24.245,21.477,-42.328
C06668=1018.446,44.257,375.405,-24.245,21.477,-42.332
C06669=1018.450,43.921,375.434,-24.244,21.478,-42.335
C06670=1018.454,43.586,375.463,-24.244,21.478,-42.339
C06671=1018.457,43.251,375.492,-24.243,21.479,-42.343
C06672=1018.460,42.916,375.520,-24.243,21.479,-42.347
C06673=1018.464,42.582,375.549,-24.242,21.479,-42.350
C06674=1018.467,42.247,375.577,-24.242,21.479,-42.354
C06675=1018.471,41.912,375.607,-24.241,21.480,-42.357
C06676=1018.474,41.577,375.635,-24.241,21.480,-42.361
C06677=1018.478,41.242,375.664,-24.240,21.481,-42.365
C06678=1018.481,40.908,375.693,-24.240,21.481,-42.369
C06679=1018.485,40.573,375.722,-24.239,21.481,-42.372
C06680=1018.488,40.238,375.751,-24.239,21.481,-42.376
C06681=1018.491,39.903,375.779,-24.238,21.482,-42.380
C06682=1018.495,39.568,375.809,-24.238,21.482,-42.383
C06683=1018.498,39.233,375.837,-24.237,21.483,-42.387
C06684=1018.501,38.899,375.866,-24.237,21.483,-42.391
C06685=1018.505,38.564,375.894,-24.236,21.483,-42.395
C06686=1018.508,38.229,375.924,-24.236,21.483,-42.398
C06687=1018.511,37.894,375.952,-24.235,21.484,-42.402
C06688=1018.515,37.559,375.980,-24.235,21.484,-42.405
C06689=1018.518,37.225,376.009,-24.234,21.485,-42.409
C06690=1018.521,36.890,376.037,-24.234,21.485,-42.413
C06691=1018.524,36.556,376.066,-24.233,21.485,-42.418
C06692=1018.528,36.220,376.095,-24.232,21.485,-42.422
C06693=1018.531,35.887,376.124,-24.232,21.486,-42.426
C06694=1018.535,35.551,376.152,-24.231,21.485,-42.429
C06695=1018.538,35.217,376.181,-24.231,21.486,-42.433
C06696=1018.541,34.882,376.210,-24.230,21.486,-42.437
C06697=1018.544,34.547,376.239,-24.230,21.487,-42.440
C06698=1018.547,34.213,376.267,-24.229,21.487,-42.444
C06699=1018.550,33.878,376.296,-24.229,21.488,-42.448
C06700=1018.553,33.543,376.324,-24.228,21.488,-42.452
C06701=1018.556,33.209,376.353,-24.228,21.489,-42.455
C06702=1018.560,32.874,376.381,-24.227,21.489,-42.459
C06703=1018.563,32.540,376.410,-24.226,21.489,-42.464
C06704=1018.565,32.205,376.438,-24.226,21.489,-42.468
C06705=1018.568,31.871,376.467,-24.225,21.489,-42.471
C06706=1018.572,31.536,376.495,-24.225,21.490,-42.475
C06707=1018.575,31.202,376.524,-24.224,21.490,-42.479
C06708=1018.578,30.867,376.552,-24.224,21.491,-42.483
C06709=1018.581,30.532,376.581,-24.223,21.491,-42.486
C06710=1018.584,30.199,376.609,-24.223,21.492,-42.490
C06711=1018.587,29.864,376.637,-24.222,21.492,-42.494
C06712=1018.590,29.529,376.666,-24.222,21.493,-42.498
C06713=1018.593,29.195,376.694,-24.221,21.492,-42.503
C06714=1018.596,28.861,376.723,-24.221,21.493,-42.507
C06715=1018.599,28.525,376.751,-24.220,21.493,-42.510
C06716=1018.601,28.191,376.780,-24.220,21.494,-42.514
C06717=1018.604,27.857,376.808,-24.219,21.494,-42.518
C06718=1018.608,27.522,376.837,-24.219,21.495,-42.522
C06719=1018.610,27.188,376.865,-24.218,21.494,-42.525
C06720=1018.613,26.854,376.893,-24.217,21.494,-42.530
C06721=1018.616,26.520,376.921,-24.217,21.495,-42.534
C06722=1018.619,26.185,376.949,-24.216,21.495,-42.538
C06723=1018.621,25.851,376.978,-24.216,21.496,-42.541
C06724=1018.624,25.516,377.007,-24.215,21.496,-42.545
C06725=1018.627,25.182,377.034,-24.215,21.497,-42.549
C06726=1018.630,24.848,377.063,-24.214,21.497,-42.553
C06727=1018.632,24.514,377.092,-24.213,21.497,-42.558
C06728=1018.636,24.186,377.119,-24.213,21.498,-42.560
C06729=1018.638,23.893,377.144,-24.213,21.498,-42.562
C06730=1018.640,23.640,377.165,-24.212,21.498,-42.565
C06731=1018.643,23.232,377.200,-24.211,21.499,-42.573
C06732=1018.646,22.823,377.234,-24.210,21.499,-42.580
C06733=1018.648,22.570,377.256,-24.210,21.500,-42.582
C06734=1018.650,22.276,377.280,-24.210,21.501,-42.584
C06735=1018.653,21.952,377.308,-24.209,21.500,-42.588
C06736=1018.656,21.595,377.337,-24.209,21.501,-42.593
C06737=1018.658,21.388,377.355,-24.208,21.501,-42.597
C06738=1018.659,21.161,377.374,-24.208,21.502,-42.599
C06739=1018.662,20.919,377.395,-24.208,21.502,-42.601
C06740=1018.664,20.671,377.416,-24.207,21.502,-42.603
C06741=1018.666,20.424,377.436,-24.207,21.502,-42.604
C06742=1018.667,20.189,377.456,-24.207,21.502,-42.608
C06743=1018.671,19.770,377.492,-24.206,21.503,-42.613
C06744=1018.673,19.423,377.521,-24.205,21.502,-42.619
C06745=1018.676,19.091,377.549,-24.205,21.503,-42.622
C06746=1018.678,18.759,377.576,-24.204,21.503,-42.626
C06747=1018.680,18.428,377.604,-24.204,21.504,-42.630
C06748=1018.683,18.097,377.632,-24.203,21.504,-42.634
C06749=1018.686,17.766,377.660,-24.202,21.504,-42.639
C06750=1018.688,17.437,377.687,-24.202,21.505,-42.643
C06751=1018.691,17.107,377.714,-24.201,21.505,-42.646
C06752=1018.693,16.778,377.742,-24.201,21.506,-42.650
C06753=1018.695,16.450,377.770,-24.200,21.506,-42.654
C06754=1018.697,16.123,377.797,-24.200,21.507,-42.658
C06755=1018.700,15.796,377.825,-24.199,21.507,-42.663
C06756=1018.703,15.469,377.852,-24.199,21.507,-42.667
C06757=1018.705,15.143,377.880,-24.198,21.508,-42.670
C06758=1018.707,14.818,377.906,-24.198,21.508,-42.674
C06759=1018.709,14.493,377.934,-24.197,21.509,-42.678
C06760=1018.712,14.169,377.961,-24.197,21.509,-42.682
C06761=1018.714,13.844,377.988,-24.196,21.509,-42.687
C06762=1018.716,13.520,378.014,-24.195,21.509,-42.691
C06763=1018.718,13.197,378.042,-24.195,21.510,-42.694
C06764=1018.721,12.872,378.068,-24.194,21.510,-42.698
C06765=1018.723,12.549,378.096,-24.194,21.511,-42.702
C06766=1018.725,12.226,378.123,-24.193,21.511,-42.707
C06767=1018.727,11.901,378.150,-24.193,21.511,-42.711
C06768=1018.729,11.579,378.176,-24.192,21.512,-42.715
C06769=1018.732,11.256,378.204,-24.192,21.512,-42.718
C06770=1018.734,10.936,378.230,-24.191,21.513,-42.722
C06771=1018.736,10.617,378.257,-24.191,21.513,-42.726
C06772=1018.738,10.300,378.283,-24.190,21.514,-42.730
C06773=1018.741,9.984,378.309,-24.190,21.514,-42.733
C06774=1018.742,9.670,378.336,-24.189,21.514,-42.738
C06775=1018.744,9.355,378.361,-24.188,21.515,-42.742
C06776=1018.746,9.040,378.388,-24.188,21.515,-42.746
C06777=1018.749,8.723,378.414,-24.187,21.516,-42.750
C06778=1018.750,8.405,378.441,-24.186,21.515,-42.755
C06779=1018.752,8.085,378.467,-24.186,21.516,-42.759
C06780=1018.754,7.761,378.494,-24.186,21.516,-42.762
C06781=1018.756,7.436,378.521,-24.185,21.517,-42.766
C06782=1018.758,7.109,378.548,-24.185,21.517,-42.770
C06783=1018.761,6.779,378.576,-24.184,21.518,-42.774
C06784=1018.762,6.451,378.603,-24.183,21.518,-42.779
C06785=1018.764,6.121,378.630,-24.183,21.518,-42.783
C06786=1018.767,5.792,378.657,-24.182,21.519,-42.786
C06787=1018.769,5.461,378.684,-24.181,21.518,-42.792
C06788=1018.770,5.130,378.712,-24.181,21.519,-42.795
C06789=1018.772,4.799,378.739,-24.180,21.519,-42.799
C06790=1018.775,4.467,378.767,-24.180,21.521,-42.803
C06791=1018.776,4.138,378.793,-24.179,21.520,-42.807
C06792=1018.778,3.824,378.819,-24.179,21.521,-42.810
C06793=1018.780,3.535,378.843,-24.179,21.521,-42.814
C06794=1018.781,3.266,378.866,-24.178,21.522,-42.818
C06795=1018.783,3.004,378.887,-24.177,21.522,-42.823
C06796=1018.785,2.735,378.909,-24.177,21.522,-42.827
C06797=1018.786,2.447,378.933,-24.176,21.523,-42.831
C06798=1018.787,2.134,378.958,-24.176,21.523,-42.834
C06799=1018.789,1.804,378.986,-24.175,21.523,-42.838
C06800=1018.791,1.471,379.013,-24.175,21.524,-42.842
C06801=1018.793,1.137,379.040,-24.174,21.525,-42.846
C06802=1018.795,0.802,379.068,-24.173,21.525,-42.851
C06803=1018.797,0.466,379.096,-24.173,21.525,-42.855
C06804=1018.798,0.129,379.124,-24.172,21.526,-42.858
C06805=1018.800,-0.210,379.152,-24.172,21.526,-42.864
C06806=1018.802,-0.550,379.179,-24.171,21.526,-42.867
C06807=1018.804,-0.892,379.207,-24.170,21.527,-42.873
C06808=1018.805,-1.235,379.236,-24.170,21.527,-42.877
C06809=1018.807,-1.580,379.264,-24.169,21.528,-42.880
C06810=1018.809,-1.927,379.292,-24.169,21.528,-42.886
C06811=1018.811,-2.275,379.320,-24.168,21.529,-42.890
C06812=1018.812,-2.625,379.350,-24.167,21.529,-42.895
C06813=1018.814,-2.976,379.378,-24.167,21.529,-42.899
C06814=1018.816,-3.329,379.407,-24.166,21.529,-42.904
C06815=1018.819,-3.683,379.436,-24.166,21.531,-42.908
C06816=1018.820,-4.040,379.465,-24.165,21.530,-42.913
C06817=1018.821,-4.402,379.495,-24.164,21.531,-42.919
C06818=1018.823,-4.768,379.525,-24.164,21.532,-42.923
C06819=1018.825,-5.139,379.554,-24.163,21.532,-42.928
C06820=1018.826,-5.512,379.585,-24.163,21.533,-42.932
C06821=1018.828,-5.887,379.615,-24.162,21.533,-42.937
C06822=1018.830,-6.262,379.646,-24.161,21.533,-42.941
C06823=1018.832,-6.637,379.677,-24.160,21.534,-42.947
C06824=1018.834,-7.009,379.707,-24.160,21.534,-42.952
C06825=1018.835,-7.379,379.737,-24.159,21.535,-42.956
C06826=1018.837,-7.745,379.767,-24.158,21.535,-42.961
C06827=1018.838,-8.108,379.796,-24.158,21.536,-42.967
C06828=1018.840,-8.471,379.826,-24.157,21.536,-42.971
C06829=1018.842,-8.834,379.855,-24.156,21.536,-42.976
C06830=1018.843,-9.196,379.885,-24.156,21.537,-42.982
C06831=1018.845,-9.558,379.914,-24.155,21.538,-42.985
C06832=1018.846,-9.919,379.943,-24.154,21.538,-42.991
C06833=1018.848,-10.280,379.973,-24.154,21.539,-42.995
C06834=1018.850,-10.641,380.001,-24.153,21.539,-43.000
C06835=1018.851,-10.999,380.030,-24.152,21.539,-43.006
C06836=1018.852,-11.358,380.060,-24.152,21.540,-43.009
C06837=1018.853,-11.713,380.088,-24.151,21.540,-43.014
C06838=1018.855,-12.068,380.116,-24.151,21.541,-43.019
C06839=1018.856,-12.422,380.145,-24.150,21.541,-43.024
C06840=1018.857,-12.774,380.174,-24.149,21.542,-43.028
C06841=1018.858,-13.125,380.202,-24.149,21.542,-43.033
C06842=1018.860,-13.473,380.230,-24.148,21.543,-43.037
C06843=1018.861,-13.819,380.258,-24.147,21.543,-43.042
C06844=1018.862,-14.164,380.286,-24.147,21.544,-43.046
C06845=1018.864,-14.505,380.313,-24.146,21.544,-43.052
C06846=1018.865,-14.845,380.341,-24.146,21.544,-43.055
C06847=1018.867,-15.183,380.368,-24.145,21.545,-43.061
C06848=1018.868,-15.520,380.394,-24.145,21.546,-43.065
C06849=1018.869,-15.855,380.422,-24.144,21.546,-43.070
C06850=1018.870,-16.189,380.448,-24.143,21.546,-43.074
C06851=1018.871,-16.523,380.475,-24.142,21.547,-43.079
C06852=1018.872,-16.856,380.502,-24.142,21.547,-43.083
C06853=1018.873,-17.189,380.529,-24.141,21.547,-43.088
C06854=1018.875,-17.522,380.556,-24.141,21.548,-43.092
C06855=1018.875,-17.887,380.584,-24.140,21.549,-43.100
C06856=1018.876,-18.109,380.602,-24.139,21.548,-43.103
C06857=1018.877,-18.357,380.622,-24.139,21.549,-43.105
C06858=1018.878,-18.618,380.643,-24.139,21.550,-43.107
C06859=1018.878,-18.880,380.664,-24.139,21.550,-43.109
C06860=1018.879,-19.128,380.684,-24.138,21.550,-43.112
C06861=1018.881,-19.544,380.717,-24.137,21.550,-43.118
C06862=1018.881,-19.716,380.731,-24.137,21.551,-43.122
C06863=1018.883,-20.049,380.757,-24.136,21.551,-43.127
C06864=1018.883,-20.382,380.784,-24.136,21.552,-43.131
C06865=1018.884,-20.715,380.811,-24.135,21.553,-43.135
C06866=1018.885,-21.047,380.837,-24.134,21.552,-43.140
C06867=1018.886,-21.381,380.864,-24.134,21.553,-43.144
C06868=1018.886,-21.713,380.890,-24.133,21.554,-43.149
C06869=1018.888,-22.047,380.917,-24.133,21.554,-43.153
C06870=1018.888,-22.379,380.943,-24.132,21.554,-43.158
C06871=1018.889,-22.712,380.970,-24.131,21.556,-43.162
C06872=1018.890,-23.045,380.996,-24.131,21.555,-43.168
C06873=1018.891,-23.377,381.023,-24.130,21.556,-43.171
C06874=1018.892,-23.710,381.049,-24.129,21.556,-43.177
C06875=1018.893,-24.043,381.075,-24.129,21.557,-43.181
C06876=1018.894,-24.376,381.102,-24.128,21.557,-43.186
C06877=1018.894,-24.708,381.128,-24.128,21.558,-43.190
C06878=1018.896,-25.041,381.155,-24.127,21.558,-43.195
C06879=1018.896,-25.374,381.181,-24.126,21.559,-43.199
C06880=1018.897,-25.707,381.207,-24.126,21.559,-43.204
C06881=1018.897,-26.039,381.233,-24.125,21.559,-43.208
C06882=1018.899,-26.372,381.260,-24.124,21.560,-43.214
C06883=1018.899,-26.705,381.286,-24.124,21.560,-43.217
C06884=1018.899,-27.038,381.313,-24.123,21.560,-43.223
C06885=1018.900,-27.371,381.338,-24.123,21.562,-43.227
C06886=1018.901,-27.704,381.365,-24.122,21.562,-43.232
C06887=1018.902,-28.036,381.391,-24.121,21.562,-43.236
C06888=1018.902,-28.369,381.418,-24.120,21.562,-43.241
C06889=1018.903,-28.702,381.443,-24.120,21.563,-43.245
C06890=1018.903,-29.035,381.470,-24.119,21.563,-43.250
C06891=1018.904,-29.367,381.496,-24.119,21.564,-43.254
C06892=1018.904,-29.700,381.522,-24.118,21.565,-43.260
C06893=1018.905,-30.033,381.548,-24.118,21.565,-43.264
C06894=1018.906,-30.365,381.574,-24.117,21.565,-43.269
C06895=1018.906,-30.698,381.600,-24.116,21.566,-43.273
C06896=1018.907,-31.030,381.627,-24.116,21.566,-43.278
C06897=1018.907,-31.364,381.653,-24.115,21.567,-43.282
C06898=1018.908,-31.697,381.679,-24.114,21.567,-43.287
C06899=1018.908,-32.029,381.705,-24.114,21.568,-43.291
C06900=1018.909,-32.362,381.731,-24.113,21.568,-43.296
C06901=1018.909,-32.695,381.757,-24.113,21.569,-43.301
C06902=1018.910,-33.027,381.783,-24.112,21.569,-43.306
C06903=1018.910,-33.360,381.809,-24.111,21.570,-43.310
C06904=1018.911,-33.692,381.836,-24.111,21.570,-43.315
C06905=1018.911,-34.025,381.861,-24.110,21.571,-43.319
C06906=1018.912,-34.358,381.887,-24.109,21.571,-43.324
C06907=1018.912,-34.690,381.913,-24.109,21.572,-43.328
C06908=1018.913,-35.023,381.939,-24.108,21.572,-43.334
C06909=1018.913,-35.357,381.966,-24.108,21.573,-43.337
C06910=1018.913,-35.689,381.991,-24.107,21.573,-43.343
C06911=1018.913,-36.022,382.017,-24.107,21.574,-43.347
C06912=1018.914,-36.354,382.043,-24.106,21.574,-43.352
C06913=1018.914,-36.687,382.069,-24.105,21.574,-43.357
C06914=1018.914,-37.020,382.094,-24.105,21.575,-43.361
C06915=1018.915,-37.352,382.121,-24.104,21.575,-43.366
C06916=1018.915,-37.685,382.146,-24.103,21.576,-43.371
C06917=1018.916,-38.018,382.172,-24.102,21.576,-43.376
C06918=1018.915,-38.350,382.198,-24.102,21.577,-43.380
C06919=1018.916,-38.682,382.224,-24.101,21.577,-43.385
C06920=1018.915,-39.016,382.249,-24.101,21.578,-43.389
C06921=1018.916,-39.348,382.275,-24.100,21.578,-43.394
C06922=1018.916,-39.681,382.301,-24.100,21.579,-43.398
C06923=1018.916,-40.014,382.327,-24.099,21.579,-43.404
C06924=1018.916,-40.346,382.352,-24.098,21.580,-43.409
C06925=1018.917,-40.678,382.379,-24.098,21.580,-43.413
C06926=1018.917,-41.011,382.404,-24.097,21.580,-43.418
C06927=1018.917,-41.344,382.430,-24.096,21.582,-43.422
C06928=1018.917,-41.676,382.456,-24.096,21.582,-43.427
C06929=1018.917,-42.009,382.481,-24.095,21.582,-43.431
C06930=1018.918,-42.341,382.507,-24.094,21.583,-43.437
C06931=1018.917,-42.674,382.533,-24.094,21.583,-43.442
C06932=1018.917,-43.007,382.558,-24.093,21.583,-43.446
C06933=1018.917,-43.339,382.584,-24.092,21.584,-43.451
C06934=1018.917,-43.672,382.610,-24.092,21.585,-43.455
C06935=1018.917,-44.005,382.635,-24.091,21.585,-43.461
C06936=1018.917,-44.337,382.661,-24.091,21.586,-43.465
C06937=1018.917,-44.670,382.686,-24.090,21.586,-43.470
C06938=1018.917,-45.002,382.711,-24.089,21.586,-43.475
C06939=1018.917,-45.334,382.738,-24.089,21.587,-43.479
C06940=1018.917,-45.667,382.762,-24.088,21.588,-43.485
C06941=1018.917,-45.999,382.788,-24.088,21.588,-43.488
C06942=1018.917,-46.332,382.813,-24.087,21.588,-43.494
C06943=1018.917,-46.664,382.839,-24.086,21.590,-43.498
C06944=1018.917,-46.997,382.865,-24.086,21.589,-43.503
C06945=1018.916,-47.330,382.890,-24.085,21.589,-43.508
C06946=1018.916,-47.662,382.916,-24.084,21.591,-43.512
C06947=1018.916,-47.995,382.941,-24.083,21.591,-43.518
C06948=1018.916,-48.327,382.966,-24.083,21.592,-43.522
C06949=1018.916,-48.660,382.992,-24.082,21.592,-43.527
C06950=1018.916,-48.992,383.017,-24.081,21.592,-43.532
C06951=1018.916,-49.325,383.043,-24.081,21.593,-43.536
C06952=1018.915,-49.657,383.068,-24.080,21.593,-43.542
C06953=1018.915,-49.989,383.093,-24.080,21.595,-43.546
C06954=1018.914,-50.322,383.118,-24.079,21.594,-43.551
C06955=1018.915,-50.654,383.143,-24.079,21.595,-43.555
C06956=1018.914,-50.987,383.169,-24.078,21.596,-43.560
C06957=1018.913,-51.318,383.194,-24.077,21.596,-43.566
C06958=1018.913,-51.651,383.219,-24.077,21.597,-43.570
C06959=1018.913,-51.983,383.245,-24.076,21.597,-43.575
C06960=1018.913,-52.316,383.270,-24.075,21.597,-43.579
C06961=1018.912,-52.648,383.295,-24.075,21.598,-43.584
C06962=1018.912,-52.980,383.321,-24.074,21.598,-43.589
C06963=1018.911,-53.313,383.345,-24.074,21.600,-43.594
C06964=1018.911,-53.645,383.371,-24.073,21.599,-43.599
C06965=1018.911,-53.977,383.396,-24.072,21.600,-43.603
C06966=1018.910,-54.310,383.421,-24.072,21.601,-43.608
C06967=1018.910,-54.642,383.446,-24.071,21.601,-43.613
C06968=1018.909,-54.974,383.471,-24.070,21.602,-43.618
C06969=1018.909,-55.307,383.496,-24.070,21.602,-43.623
C06970=1018.908,-55.639,383.521,-24.069,21.603,-43.627
C06971=1018.908,-55.973,383.546,-24.068,21.603,-43.632
C06972=1018.908,-56.305,383.572,-24.068,21.603,-43.637
C06973=1018.906,-56.638,383.597,-24.067,21.605,-43.642
C06974=1018.907,-56.971,383.622,-24.066,21.604,-43.647
C06975=1018.906,-57.305,383.646,-24.066,21.605,-43.652
C06976=1018.905,-57.639,383.672,-24.065,21.606,-43.656
C06977=1018.905,-57.974,383.696,-24.064,21.606,-43.662
C06978=1018.904,-58.308,383.722,-24.064,21.607,-43.666
C06979=1018.903,-58.643,383.747,-24.063,21.607,-43.671
C06980=1018.903,-58.978,383.773,-24.062,21.608,-43.676
C06981=1018.902,-59.314,383.797,-24.062,21.608,-43.680
C06982=1018.902,-59.649,383.823,-24.061,21.609,-43.686
C06983=1018.901,-59.986,383.848,-24.060,21.609,-43.691
C06984=1018.900,-60.323,383.873,-24.060,21.610,-43.695
C06985=1018.899,-60.661,383.898,-24.059,21.610,-43.700
C06986=1018.899,-60.998,383.924,-24.059,21.611,-43.706
C06987=1018.898,-61.336,383.949,-24.058,21.611,-43.710
C06988=1018.897,-61.675,383.974,-24.057,21.612,-43.715
C06989=1018.897,-62.013,384.000,-24.057,21.612,-43.720
C06990=1018.895,-62.353,384.025,-24.056,21.614,-43.725
C06991=1018.895,-62.692,384.050,-24.055,21.613,-43.730
C06992=1018.894,-63.033,384.076,-24.055,21.614,-43.735
C06993=1018.893,-63.372,384.100,-24.054,21.615,-43.739
C06994=1018.892,-63.713,384.126,-24.053,21.616,-43.745
C06995=1018.892,-64.055,384.152,-24.053,21.615,-43.750
C06996=1018.891,-64.395,384.177,-24.052,21.617,-43.754
C06997=1018.890,-64.736,384.202,-24.051,21.617,-43.759
C06998=1018.889,-65.078,384.227,-24.051,21.618,-43.765
C06999=1018.888,-65.421,384.254,-24.050,21.617,-43.770
C07000=1018.887,-65.763,384.278,-24.050,21.619,-43.774
C07001=1018.886,-66.105,384.304,-24.049,21.619,-43.780
C07002=1018.885,-66.449,384.330,-24.048,21.620,-43.785
C07003=1018.884,-66.792,384.354,-24.048,21.620,-43.789
C07004=1018.883,-67.134,384.380,-24.047,21.621,-43.795
C07005=1018.882,-67.477,384.406,-24.046,21.621,-43.800
C07006=1018.880,-67.821,384.431,-24.045,21.622,-43.805
C07007=1018.880,-68.165,384.456,-24.045,21.622,-43.809
C07008=1018.879,-68.509,384.481,-24.044,21.623,-43.815
C07009=1018.878,-68.853,384.507,-24.043,21.623,-43.820
C07010=1018.877,-69.196,384.533,-24.043,21.624,-43.824
C07011=1018.876,-69.541,384.558,-24.042,21.624,-43.829
C07012=1018.874,-69.884,384.583,-24.041,21.625,-43.835
C07013=1018.873,-70.228,384.609,-24.041,21.625,-43.840
C07014=1018.872,-70.573,384.634,-24.040,21.626,-43.844
C07015=1018.871,-70.916,384.659,-24.040,21.627,-43.850
C07016=1018.870,-71.260,384.684,-24.039,21.627,-43.855
C07017=1018.868,-71.604,384.709,-24.038,21.628,-43.861
C07018=1018.867,-71.948,384.735,-24.038,21.628,-43.865
C07019=1018.866,-72.293,384.760,-24.037,21.629,-43.870
C07020=1018.865,-72.637,384.786,-24.036,21.629,-43.875
C07021=1018.863,-72.981,384.810,-24.035,21.630,-43.881
C07022=1018.862,-73.324,384.836,-24.035,21.630,-43.885
C07023=1018.860,-73.668,384.861,-24.034,21.631,-43.890
C07024=1018.859,-74.012,384.886,-24.033,21.632,-43.896
C07025=1018.858,-74.355,384.911,-24.033,21.632,-43.901
C07026=1018.857,-74.699,384.937,-24.032,21.633,-43.905
C07027=1018.855,-75.042,384.961,-24.031,21.633,-43.911
C07028=1018.854,-75.385,384.986,-24.031,21.634,-43.916
C07029=1018.852,-75.729,385.011,-24.030,21.634,-43.920
C07030=1018.851,-76.072,385.036,-24.030,21.635,-43.926
C07031=1018.850,-76.413,385.061,-24.029,21.635,-43.931
C07032=1018.848,-76.756,385.086,-24.028,21.636,-43.936
C07033=1018.847,-77.099,385.111,-24.028,21.636,-43.940
C07034=1018.846,-77.440,385.136,-24.027,21.637,-43.946
C07035=1018.844,-77.782,385.161,-24.026,21.637,-43.951
C07036=1018.843,-78.123,385.186,-24.026,21.639,-43.955
C07037=1018.841,-78.465,385.210,-24.025,21.638,-43.960
C07038=1018.839,-78.806,385.235,-24.024,21.639,-43.966
C07039=1018.838,-79.146,385.260,-24.023,21.639,-43.971
C07040=1018.836,-79.486,385.285,-24.023,21.641,-43.975
C07041=1018.835,-79.826,385.309,-24.022,21.641,-43.981
C07042=1018.833,-80.166,385.335,-24.021,21.641,-43.986
C07043=1018.831,-80.504,385.358,-24.021,21.643,-43.990
C07044=1018.830,-80.843,385.382,-24.020,21.643,-43.995
C07045=1018.828,-81.181,385.407,-24.020,21.643,-44.001
C07046=1018.826,-81.519,385.431,-24.019,21.644,-44.005
C07047=1018.825,-81.857,385.456,-24.018,21.645,-44.010
C07048=1018.823,-82.194,385.481,-24.018,21.645,-44.016
C07049=1018.821,-82.530,385.505,-24.017,21.645,-44.021
C07050=1018.819,-82.865,385.529,-24.016,21.646,-44.025
C07051=1018.818,-83.201,385.553,-24.016,21.647,-44.031
C07052=1018.816,-83.537,385.577,-24.015,21.647,-44.036
C07053=1018.814,-83.872,385.601,-24.015,21.648,-44.040
C07054=1018.813,-84.206,385.625,-24.014,21.648,-44.045
C07055=1018.811,-84.556,385.651,-24.013,21.649,-44.051
C07056=1018.808,-84.953,385.679,-24.012,21.650,-44.056
C07057=1018.808,-85.165,385.694,-24.012,21.649,-44.060
C07058=1018.806,-85.379,385.709,-24.012,21.649,-44.062
C07059=1018.804,-85.788,385.738,-24.011,21.650,-44.067
C07060=1018.803,-86.147,385.765,-24.010,21.651,-44.073
C07061=1018.800,-86.476,385.788,-24.009,21.652,-44.078
C07062=1018.799,-86.798,385.810,-24.009,21.652,-44.082
C07063=1018.796,-87.115,385.834,-24.008,21.653,-44.088
C07064=1018.795,-87.427,385.856,-24.007,21.653,-44.093
C07065=1018.793,-87.738,385.879,-24.007,21.654,-44.097
C07066=1018.791,-88.051,385.901,-24.006,21.654,-44.102
C07067=1018.789,-88.369,385.923,-24.006,21.655,-44.106
C07068=1018.787,-88.740,385.950,-24.005,21.656,-44.114
C07069=1018.786,-88.959,385.965,-24.004,21.656,-44.117
C07070=1018.784,-89.193,385.983,-24.004,21.656,-44.119
C07071=1018.783,-89.431,385.999,-24.004,21.656,-44.121
C07072=1018.782,-89.663,386.016,-24.004,21.657,-44.123
C07073=1018.779,-90.068,386.045,-24.003,21.658,-44.130
C07074=1018.778,-90.406,386.068,-24.002,21.658,-44.136
C07075=1018.775,-90.736,386.092,-24.001,21.659,-44.141
C07076=1018.773,-91.065,386.116,-24.001,21.660,-44.145
C07077=1018.771,-91.394,386.139,-24.000,21.660,-44.150
C07078=1018.769,-91.722,386.162,-23.999,21.660,-44.156
C07079=1018.767,-92.050,386.186,-23.999,21.661,-44.160
C07080=1018.764,-92.377,386.209,-23.998,21.662,-44.165
C07081=1018.763,-92.704,386.232,-23.998,21.662,-44.169
C07082=1018.761,-93.030,386.255,-23.997,21.663,-44.175
C07083=1018.759,-93.355,386.278,-23.996,21.663,-44.180
C07084=1018.756,-93.681,386.300,-23.996,21.664,-44.184
C07085=1018.754,-94.005,386.324,-23.995,21.664,-44.189
C07086=1018.752,-94.330,386.346,-23.994,21.665,-44.193
C07087=1018.749,-94.653,386.369,-23.994,21.666,-44.199
C07088=1018.747,-94.975,386.392,-23.993,21.666,-44.204
C07089=1018.745,-95.299,386.415,-23.993,21.666,-44.207
C07090=1018.743,-95.621,386.438,-23.992,21.667,-44.213
C07091=1018.741,-95.942,386.460,-23.991,21.668,-44.217
C07092=1018.739,-96.264,386.483,-23.991,21.668,-44.222
C07093=1018.737,-96.586,386.506,-23.990,21.669,-44.226
C07094=1018.735,-96.907,386.528,-23.989,21.669,-44.231
C07095=1018.732,-97.228,386.551,-23.989,21.670,-44.236
C07096=1018.729,-97.549,386.573,-23.988,21.670,-44.241
C07097=1018.727,-97.870,386.596,-23.987,21.670,-44.246
C07098=1018.725,-98.191,386.618,-23.987,21.672,-44.250
C07099=1018.722,-98.511,386.641,-23.986,21.671,-44.255
C07100=1018.720,-98.833,386.663,-23.986,21.673,-44.260
C07101=1018.718,-99.153,386.686,-23.985,21.673,-44.265
C07102=1018.715,-99.475,386.709,-23.985,21.673,-44.268
C07103=1018.713,-99.796,386.731,-23.984,21.674,-44.274
C07104=1018.711,-100.118,386.754,-23.983,21.675,-44.278
C07105=1018.708,-100.441,386.776,-23.983,21.675,-44.283
C07106=1018.706,-100.763,386.798,-23.982,21.676,-44.287
C07107=1018.703,-101.086,386.821,-23.981,21.676,-44.292
C07108=1018.701,-101.410,386.844,-23.981,21.677,-44.298
C07109=1018.698,-101.734,386.867,-23.980,21.677,-44.302
C07110=1018.696,-102.058,386.889,-23.980,21.678,-44.307
C07111=1018.693,-102.384,386.912,-23.979,21.679,-44.311
C07112=1018.690,-102.709,386.934,-23.978,21.679,-44.316
C07113=1018.688,-103.035,386.957,-23.978,21.680,-44.320
C07114=1018.686,-103.362,386.980,-23.977,21.680,-44.326
C07115=1018.683,-103.689,387.002,-23.976,21.681,-44.331
C07116=1018.680,-104.016,387.025,-23.976,21.681,-44.335
C07117=1018.677,-104.343,387.048,-23.975,21.681,-44.340
C07118=1018.674,-104.672,387.071,-23.975,21.683,-44.344
C07119=1018.672,-105.000,387.094,-23.974,21.683,-44.350
C07120=1018.669,-105.328,387.116,-23.974,21.684,-44.354
C07121=1018.666,-105.657,387.139,-23.973,21.684,-44.359
C07122=1018.664,-105.986,387.162,-23.972,21.685,-44.365
C07123=1018.661,-106.315,387.184,-23.972,21.685,-44.368
C07124=1018.658,-106.644,387.207,-23.971,21.685,-44.374
C07125=1018.655,-106.973,387.231,-23.971,21.687,-44.378
C07126=1018.652,-107.302,387.254,-23.970,21.687,-44.383
C07127=1018.650,-107.631,387.275,-23.969,21.687,-44.388
C07128=1018.647,-107.959,387.298,-23.969,21.688,-44.392
C07129=1018.644,-108.288,387.321,-23.968,21.689,-44.398
C07130=1018.642,-108.618,387.343,-23.967,21.689,-44.402
C07131=1018.638,-108.947,387.367,-23.967,21.689,-44.407
C07132=1018.635,-109.275,387.389,-23.966,21.690,-44.412
C07133=1018.632,-109.604,387.412,-23.965,21.691,-44.416
C07134=1018.630,-109.933,387.434,-23.965,21.691,-44.422
C07135=1018.627,-110.262,387.457,-23.964,21.692,-44.426
C07136=1018.624,-110.591,387.480,-23.963,21.692,-44.431
C07137=1018.621,-110.919,387.503,-23.963,21.693,-44.436
C07138=1018.617,-111.248,387.526,-23.962,21.693,-44.440
C07139=1018.614,-111.578,387.548,-23.962,21.694,-44.446
C07140=1018.611,-111.906,387.570,-23.961,21.695,-44.449
C07141=1018.608,-112.235,387.593,-23.960,21.695,-44.455
C07142=1018.605,-112.563,387.615,-23.960,21.696,-44.459
C07143=1018.602,-112.892,387.638,-23.959,21.696,-44.464
C07144=1018.599,-113.221,387.660,-23.958,21.697,-44.470
C07145=1018.596,-113.549,387.682,-23.958,21.697,-44.473
C07146=1018.593,-113.878,387.705,-23.957,21.698,-44.479
C07147=1018.590,-114.207,387.728,-23.957,21.699,-44.483
C07148=1018.586,-114.535,387.750,-23.956,21.699,-44.488
C07149=1018.583,-114.863,387.773,-23.956,21.700,-44.492
C07150=1018.580,-115.192,387.795,-23.955,21.700,-44.497
C07151=1018.576,-115.520,387.817,-23.954,21.701,-44.503
C07152=1018.573,-115.849,387.839,-23.954,21.701,-44.507
C07153=1018.570,-116.178,387.862,-23.953,21.701,-44.512
C07154=1018.567,-116.506,387.884,-23.953,21.703,-44.516
C07155=1018.564,-116.835,387.907,-23.952,21.703,-44.521
C07156=1018.560,-117.163,387.929,-23.951,21.704,-44.525
C07157=1018.557,-117.492,387.952,-23.951,21.704,-44.531
C07158=1018.553,-117.820,387.974,-23.950,21.705,-44.535
C07159=1018.550,-118.148,387.997,-23.949,21.705,-44.540
C07160=1018.546,-118.477,388.019,-23.949,21.705,-44.545
C07161=1018.543,-118.805,388.041,-23.948,21.707,-44.549
C07162=1018.539,-119.133,388.063,-23.948,21.707,-44.554
C07163=1018.536,-119.462,388.086,-23.947,21.707,-44.558
C07164=1018.533,-119.790,388.108,-23.946,21.708,-44.564
C07165=1018.529,-120.118,388.130,-23.946,21.709,-44.568
C07166=1018.526,-120.446,388.152,-23.945,21.709,-44.573
C07167=1018.523,-120.775,388.175,-23.945,21.710,-44.577
C07168=1018.519,-121.104,388.196,-23.944,21.710,-44.582
C07169=1018.515,-121.432,388.218,-23.944,21.711,-44.586
C07170=1018.512,-121.760,388.240,-23.943,21.711,-44.591
C07171=1018.508,-122.089,388.263,-23.942,21.712,-44.597
C07172=1018.505,-122.417,388.285,-23.942,21.713,-44.601
C07173=1018.500,-122.806,388.312,-23.941,21.713,-44.606
C07174=1018.497,-123.104,388.332,-23.940,21.714,-44.610
C07175=1018.494,-123.401,388.351,-23.940,21.714,-44.615
C07176=1018.490,-123.729,388.373,-23.939,21.715,-44.620
C07177=1018.486,-124.057,388.395,-23.939,21.715,-44.625
C07178=1018.483,-124.386,388.417,-23.938,21.716,-44.628
C07179=1018.479,-124.714,388.440,-23.937,21.717,-44.634
C07180=1018.475,-125.042,388.462,-23.937,21.717,-44.638
C07181=1018.471,-125.370,388.484,-23.936,21.717,-44.643
C07182=1018.467,-125.698,388.507,-23.936,21.719,-44.647
C07183=1018.463,-126.026,388.529,-23.935,21.719,-44.652
C07184=1018.460,-126.355,388.551,-23.935,21.720,-44.657
C07185=1018.457,-126.682,388.572,-23.934,21.720,-44.662
C07186=1018.453,-127.010,388.595,-23.933,21.720,-44.667
C07187=1018.448,-127.338,388.616,-23.933,21.721,-44.671
C07188=1018.444,-127.667,388.638,-23.932,21.721,-44.676
C07189=1018.441,-127.995,388.660,-23.931,21.722,-44.680
C07190=1018.437,-128.323,388.682,-23.931,21.723,-44.686
C07191=1018.432,-128.651,388.704,-23.930,21.723,-44.689
C07192=1018.429,-128.979,388.726,-23.929,21.723,-44.695
C07193=1018.425,-129.307,388.748,-23.929,21.725,-44.699
C07194=1018.421,-129.635,388.769,-23.928,21.724,-44.704
C07195=1018.417,-129.963,388.791,-23.928,21.726,-44.708
C07196=1018.413,-130.291,388.813,-23.927,21.726,-44.713
C07197=1018.409,-130.619,388.835,-23.927,21.726,-44.717
C07198=1018.405,-130.947,388.857,-23.926,21.727,-44.723
C07199=1018.401,-131.275,388.879,-23.926,21.728,-44.726
C07200=1018.397,-131.603,388.901,-23.925,21.728,-44.732
C07201=1018.392,-131.931,388.923,-23.924,21.729,-44.736
C07202=1018.388,-132.259,388.945,-23.924,21.729,-44.741
C07203=1018.384,-132.587,388.966,-23.923,21.730,-44.745
C07204=1018.381,-132.915,388.988,-23.922,21.731,-44.750
C07205=1018.376,-133.243,389.010,-23.922,21.731,-44.754
C07206=1018.372,-133.571,389.032,-23.921,21.731,-44.759
C07207=1018.368,-133.899,389.053,-23.921,21.732,-44.763
C07208=1018.747,-133.871,388.816,-23.921,21.732,-44.763
C07209=1018.752,-133.543,388.795,-23.921,21.731,-44.759
C07210=1018.755,-133.216,388.773,-23.922,21.731,-44.754
C07211=1018.760,-132.888,388.752,-23.922,21.731,-44.750
C07212=1018.763,-132.560,388.730,-23.923,21.730,-44.745
C07213=1018.768,-132.232,388.708,-23.924,21.729,-44.741
C07214=1018.772,-131.903,388.686,-23.924,21.729,-44.736
C07215=1018.776,-131.575,388.664,-23.925,21.728,-44.732
C07216=1018.779,-131.248,388.643,-23.926,21.728,-44.726
C07217=1018.784,-130.920,388.621,-23.926,21.727,-44.723
C07218=1018.788,-130.592,388.599,-23.927,21.726,-44.717
C07219=1018.792,-130.264,388.578,-23.927,21.726,-44.713
C07220=1018.796,-129.935,388.555,-23.928,21.726,-44.708
C07221=1018.800,-129.607,388.533,-23.928,21.724,-44.704
C07222=1018.804,-129.280,388.512,-23.929,21.725,-44.699
C07223=1018.807,-128.952,388.490,-23.929,21.723,-44.695
C07224=1018.811,-128.623,388.468,-23.930,21.723,-44.689
C07225=1018.815,-128.295,388.446,-23.931,21.723,-44.686
C07226=1018.819,-127.967,388.424,-23.931,21.722,-44.680
C07227=1018.823,-127.639,388.402,-23.932,21.721,-44.676
C07228=1018.826,-127.312,388.381,-23.933,21.721,-44.671
C07229=1018.830,-126.983,388.358,-23.933,21.720,-44.667
C07230=1018.834,-126.655,388.336,-23.934,21.720,-44.662
C07231=1018.838,-126.327,388.314,-23.935,21.720,-44.657
C07232=1018.842,-125.999,388.293,-23.935,21.719,-44.652
C07233=1018.846,-125.671,388.271,-23.936,21.719,-44.647
C07234=1018.849,-125.343,388.249,-23.936,21.717,-44.643
C07235=1018.853,-125.015,388.227,-23.937,21.717,-44.638
C07236=1018.857,-124.687,388.205,-23.937,21.717,-44.634
C07237=1018.861,-124.358,388.183,-23.938,21.716,-44.628
C07238=1018.864,-124.030,388.161,-23.939,21.715,-44.625
C07239=1018.868,-123.702,388.138,-23.939,21.715,-44.620
C07240=1018.871,-123.374,388.116,-23.940,21.714,-44.615
C07241=1018.874,-123.046,388.094,-23.940,21.714,-44.610
C07242=1018.878,-122.717,388.072,-23.941,21.713,-44.606
C07243=1018.882,-122.389,388.050,-23.942,21.713,-44.601
C07244=1018.886,-122.061,388.028,-23.942,21.712,-44.597
C07245=1018.889,-121.733,388.006,-23.943,21.711,-44.591
C07246=1018.892,-121.405,387.983,-23.944,21.711,-44.586
C07247=1018.895,-121.076,387.962,-23.944,21.710,-44.582
C07248=1018.899,-120.748,387.940,-23.945,21.710,-44.577
C07249=1018.903,-120.419,387.918,-23.945,21.709,-44.573
C07250=1018.906,-120.091,387.895,-23.946,21.709,-44.568
C07251=1018.910,-119.763,387.873,-23.946,21.708,-44.564
C07252=1018.913,-119.434,387.851,-23.947,21.707,-44.558
C07253=1018.916,-119.106,387.828,-23.948,21.707,-44.554
C07254=1018.920,-118.778,387.806,-23.948,21.707,-44.549
C07255=1018.923,-118.450,387.784,-23.949,21.705,-44.545
C07256=1018.926,-118.121,387.762,-23.949,21.705,-44.540
C07257=1018.929,-117.793,387.739,-23.950,21.705,-44.535
C07258=1018.933,-117.464,387.717,-23.951,21.704,-44.531
C07259=1018.936,-117.135,387.695,-23.951,21.704,-44.525
C07260=1018.940,-116.807,387.673,-23.952,21.703,-44.521
C07261=1018.943,-116.479,387.650,-23.953,21.703,-44.516
C07262=1018.947,-116.150,387.628,-23.953,21.701,-44.512
C07263=1018.950,-115.822,387.605,-23.954,21.701,-44.507
C07264=1018.953,-115.493,387.582,-23.954,21.701,-44.503
C07265=1018.956,-115.166,387.561,-23.955,21.700,-44.497
C07266=1018.959,-114.836,387.539,-23.956,21.700,-44.492
C07267=1018.962,-114.508,387.516,-23.956,21.699,-44.488
C07268=1018.965,-114.179,387.493,-23.957,21.699,-44.483
C07269=1018.968,-113.851,387.471,-23.957,21.698,-44.479
C07270=1018.971,-113.522,387.449,-23.958,21.697,-44.473
C07271=1018.974,-113.193,387.427,-23.958,21.697,-44.470
C07272=1018.977,-112.865,387.404,-23.959,21.696,-44.464
C07273=1018.980,-112.536,387.381,-23.960,21.696,-44.459
C07274=1018.983,-112.208,387.358,-23.960,21.695,-44.455
C07275=1018.986,-111.879,387.336,-23.961,21.695,-44.449
C07276=1018.989,-111.550,387.314,-23.962,21.694,-44.446
C07277=1018.992,-111.221,387.291,-23.962,21.693,-44.440
C07278=1018.995,-110.893,387.268,-23.963,21.693,-44.436
C07279=1018.999,-110.563,387.245,-23.963,21.692,-44.431
C07280=1019.001,-110.234,387.223,-23.964,21.692,-44.426
C07281=1019.004,-109.906,387.201,-23.965,21.691,-44.422
C07282=1019.008,-109.577,387.178,-23.965,21.691,-44.416
C07283=1019.011,-109.248,387.155,-23.966,21.690,-44.412
C07284=1019.013,-108.919,387.133,-23.967,21.689,-44.407
C07285=1019.016,-108.590,387.110,-23.967,21.689,-44.402
C07286=1019.019,-108.262,387.087,-23.968,21.689,-44.398
C07287=1019.021,-107.933,387.065,-23.969,21.688,-44.392
C07288=1019.025,-107.603,387.042,-23.969,21.687,-44.388
C07289=1019.027,-107.274,387.019,-23.970,21.687,-44.383
C07290=1019.030,-106.945,386.997,-23.971,21.687,-44.378
C07291=1019.033,-106.617,386.974,-23.971,21.685,-44.374
C07292=1019.035,-106.288,386.951,-23.972,21.685,-44.368
C07293=1019.038,-105.959,386.928,-23.972,21.685,-44.365
C07294=1019.041,-105.630,386.906,-23.973,21.684,-44.359
C07295=1019.043,-105.301,386.883,-23.974,21.684,-44.354
C07296=1019.046,-104.973,386.860,-23.974,21.683,-44.350
C07297=1019.049,-104.644,386.838,-23.975,21.683,-44.344
C07298=1019.052,-104.317,386.815,-23.975,21.681,-44.340
